LIN {X 74.035,Y -43.514,Z -167.127,A -90.000,B 90.000,C 0.000} C_DIS
LIN {X 73.239,Y -43.520,Z -169.410,A -90.000,B 90.000,C 0.000} C_DIS
LIN {X 72.844,Y -43.519,Z -170.536,A -90.000,B 90.000,C 0.000} C_DIS
LIN {X 72.299,Y -43.524,Z -172.033,A -90.000,B 90.000,C 0.000} C_DIS
LIN {X 72.099,Y -43.529,Z -172.557,A -90.000,B 90.000,C 0.000} C_DIS
LIN {X 71.692,Y -43.549,Z -173.637,A -90.000,B 90.000,C 0.000} C_DIS
LIN {X 71.059,Y -43.555,Z -175.551,A -90.000,B 90.000,C 0.000} C_DIS
LIN {X 70.896,Y -43.570,Z -176.056,A -90.000,B 90.000,C 0.000} C_DIS
LIN {X 70.529,Y -43.551,Z -177.830,A -90.000,B 90.000,C 0.000} C_DIS
LIN {X 70.400,Y -43.548,Z -178.399,A -90.000,B 90.000,C 0.000} C_DIS
LIN {X 70.060,Y -43.525,Z -180.717,A -90.000,B 90.000,C 0.000} C_DIS
LIN {X 70.039,Y -43.519,Z -180.942,A -90.000,B 90.000,C 0.000} C_DIS
LIN {X 69.857,Y -43.488,Z -182.943,A -90.000,B 90.000,C 0.000} C_DIS
LIN {X 69.817,Y -43.471,Z -183.612,A -90.000,B 90.000,C 0.000} C_DIS
LIN {X 69.805,Y -43.466,Z -183.813,A -90.000,B 90.000,C 0.000} C_DIS
LIN {X 69.642,Y -43.421,Z -186.238,A -90.000,B 90.000,C 0.000} C_DIS
LIN {X 69.579,Y -43.400,Z -187.145,A -90.000,B 90.000,C 0.000} C_DIS
LIN {X 69.514,Y -43.379,Z -188.002,A -90.000,B 90.000,C 0.000} C_DIS
LIN {X 69.477,Y -43.368,Z -188.428,A -90.000,B 90.000,C 0.000} C_DIS
LIN {X 69.418,Y -43.357,Z -188.971,A -90.000,B 90.000,C 0.000} C_DIS
LIN {X 69.299,Y -43.324,Z -190.039,A -90.000,B 90.000,C 0.000} C_DIS
LIN {X 69.261,Y -43.308,Z -190.358,A -90.000,B 90.000,C 0.000} C_DIS
LIN {X 69.261,Y -60.000,Z -190.358,A -90.000,B 90.000,C 0.000} C_DIS
LIN {X 59.148,Y -60.000,Z -133.648,A -90.000,B 90.000,C 0.000} C_DIS
LIN {X 59.148,Y -43.308,Z -133.648,A -90.000,B 90.000,C 0.000} C_DIS
LIN {X 59.314,Y -43.330,Z -133.579,A -90.000,B 90.000,C 0.000} C_DIS
LIN {X 59.672,Y -43.381,Z -133.445,A -90.000,B 90.000,C 0.000} C_DIS
LIN {X 60.638,Y -43.533,Z -133.112,A -90.000,B 90.000,C 0.000} C_DIS
LIN {X 61.670,Y -43.677,Z -132.764,A -90.000,B 90.000,C 0.000} C_DIS
LIN {X 61.820,Y -43.698,Z -132.716,A -90.000,B 90.000,C 0.000} C_DIS
LIN {X 61.951,Y -43.718,Z -132.678,A -90.000,B 90.000,C 0.000} C_DIS
LIN {X 62.168,Y -43.758,Z -132.615,A -90.000,B 90.000,C 0.000} C_DIS
LIN {X 62.369,Y -43.796,Z -132.562,A -90.000,B 90.000,C 0.000} C_DIS
LIN {X 62.552,Y -43.831,Z -132.519,A -90.000,B 90.000,C 0.000} C_DIS
LIN {X 62.943,Y -43.909,Z -132.439,A -90.000,B 90.000,C 0.000} C_DIS
LIN {X 63.093,Y -43.940,Z -132.412,A -90.000,B 90.000,C 0.000} C_DIS
LIN {X 63.216,Y -43.967,Z -132.392,A -90.000,B 90.000,C 0.000} C_DIS
LIN {X 63.328,Y -43.991,Z -132.378,A -90.000,B 90.000,C 0.000} C_DIS
LIN {X 63.581,Y -44.028,Z -132.352,A -90.000,B 90.000,C 0.000} C_DIS
LIN {X 63.758,Y -44.054,Z -132.339,A -90.000,B 90.000,C 0.000} C_DIS
LIN {X 64.159,Y -44.115,Z -132.327,A -90.000,B 90.000,C 0.000} C_DIS
LIN {X 64.303,Y -44.138,Z -132.327,A -90.000,B 90.000,C 0.000} C_DIS
LIN {X 65.331,Y -44.306,Z -132.343,A -90.000,B 90.000,C 0.000} C_DIS
LIN {X 65.660,Y -44.358,Z -132.351,A -90.000,B 90.000,C 0.000} C_DIS
LIN {X 65.799,Y -44.369,Z -132.355,A -90.000,B 90.000,C 0.000} C_DIS
LIN {X 65.974,Y -44.379,Z -132.361,A -90.000,B 90.000,C 0.000} C_DIS
LIN {X 66.177,Y -44.391,Z -132.376,A -90.000,B 90.000,C 0.000} C_DIS
LIN {X 66.618,Y -44.418,Z -132.426,A -90.000,B 90.000,C 0.000} C_DIS
LIN {X 66.734,Y -44.426,Z -132.443,A -90.000,B 90.000,C 0.000} C_DIS
LIN {X 67.191,Y -44.459,Z -132.526,A -90.000,B 90.000,C 0.000} C_DIS
LIN {X 67.404,Y -44.474,Z -132.567,A -90.000,B 90.000,C 0.000} C_DIS
LIN {X 67.694,Y -44.496,Z -132.633,A -90.000,B 90.000,C 0.000} C_DIS
LIN {X 67.883,Y -44.509,Z -132.684,A -90.000,B 90.000,C 0.000} C_DIS
LIN {X 68.117,Y -44.524,Z -132.758,A -90.000,B 90.000,C 0.000} C_DIS
LIN {X 68.235,Y -44.524,Z -132.797,A -90.000,B 90.000,C 0.000} C_DIS
LIN {X 69.600,Y -44.469,Z -133.270,A -90.000,B 90.000,C 0.000} C_DIS
LIN {X 69.759,Y -44.463,Z -133.330,A -90.000,B 90.000,C 0.000} C_DIS
LIN {X 70.074,Y -44.451,Z -133.459,A -90.000,B 90.000,C 0.000} C_DIS
LIN {X 70.309,Y -44.443,Z -133.564,A -90.000,B 90.000,C 0.000} C_DIS
LIN {X 70.481,Y -44.437,Z -133.650,A -90.000,B 90.000,C 0.000} C_DIS
LIN {X 70.755,Y -44.429,Z -133.798,A -90.000,B 90.000,C 0.000} C_DIS
LIN {X 70.990,Y -44.420,Z -133.930,A -90.000,B 90.000,C 0.000} C_DIS
LIN {X 71.077,Y -44.411,Z -133.981,A -90.000,B 90.000,C 0.000} C_DIS
LIN {X 71.147,Y -44.402,Z -134.025,A -90.000,B 90.000,C 0.000} C_DIS
LIN {X 71.340,Y -44.376,Z -134.152,A -90.000,B 90.000,C 0.000} C_DIS
LIN {X 71.676,Y -44.334,Z -134.389,A -90.000,B 90.000,C 0.000} C_DIS
LIN {X 71.836,Y -44.314,Z -134.512,A -90.000,B 90.000,C 0.000} C_DIS
LIN {X 72.068,Y -44.286,Z -134.700,A -90.000,B 90.000,C 0.000} C_DIS
LIN {X 72.330,Y -44.255,Z -134.922,A -90.000,B 90.000,C 0.000} C_DIS
LIN {X 72.460,Y -44.240,Z -135.039,A -90.000,B 90.000,C 0.000} C_DIS
LIN {X 72.525,Y -44.233,Z -135.101,A -90.000,B 90.000,C 0.000} C_DIS
LIN {X 72.757,Y -44.206,Z -135.333,A -90.000,B 90.000,C 0.000} C_DIS
LIN {X 73.431,Y -44.132,Z -136.043,A -90.000,B 90.000,C 0.000} C_DIS
LIN {X 73.613,Y -44.113,Z -136.246,A -90.000,B 90.000,C 0.000} C_DIS
LIN {X 73.667,Y -44.107,Z -136.309,A -90.000,B 90.000,C 0.000} C_DIS
LIN {X 73.937,Y -44.080,Z -136.639,A -90.000,B 90.000,C 0.000} C_DIS
LIN {X 74.056,Y -44.065,Z -136.797,A -90.000,B 90.000,C 0.000} C_DIS
LIN {X 74.241,Y -44.043,Z -137.053,A -90.000,B 90.000,C 0.000} C_DIS
LIN {X 74.346,Y -44.031,Z -137.211,A -90.000,B 90.000,C 0.000} C_DIS
LIN {X 74.417,Y -44.017,Z -137.322,A -90.000,B 90.000,C 0.000} C_DIS
LIN {X 74.552,Y -43.991,Z -137.546,A -90.000,B 90.000,C 0.000} C_DIS
LIN {X 74.951,Y -43.916,Z -138.254,A -90.000,B 90.000,C 0.000} C_DIS
LIN {X 75.488,Y -43.810,Z -139.094,A -90.000,B 90.000,C 0.000} C_DIS
LIN {X 75.587,Y -43.791,Z -139.263,A -90.000,B 90.000,C 0.000} C_DIS
LIN {X 75.716,Y -43.767,Z -139.493,A -90.000,B 90.000,C 0.000} C_DIS
LIN {X 75.863,Y -43.740,Z -139.772,A -90.000,B 90.000,C 0.000} C_DIS
LIN {X 76.002,Y -43.711,Z -140.057,A -90.000,B 90.000,C 0.000} C_DIS
LIN {X 76.088,Y -43.694,Z -140.251,A -90.000,B 90.000,C 0.000} C_DIS
LIN {X 76.773,Y -43.558,Z -141.907,A -90.000,B 90.000,C 0.000} C_DIS
LIN {X 76.859,Y -43.541,Z -142.139,A -90.000,B 90.000,C 0.000} C_DIS
LIN {X 77.001,Y -43.514,Z -142.567,A -90.000,B 90.000,C 0.000} C_DIS
LIN {X 77.079,Y -43.501,Z -142.832,A -90.000,B 90.000,C 0.000} C_DIS
LIN {X 77.166,Y -43.485,Z -143.164,A -90.000,B 90.000,C 0.000} C_DIS
LIN {X 77.257,Y -43.465,Z -143.511,A -90.000,B 90.000,C 0.000} C_DIS
LIN {X 77.395,Y -43.429,Z -144.052,A -90.000,B 90.000,C 0.000} C_DIS
LIN {X 77.452,Y -43.415,Z -144.315,A -90.000,B 90.000,C 0.000} C_DIS
LIN {X 77.497,Y -43.400,Z -144.536,A -90.000,B 90.000,C 0.000} C_DIS
LIN {X 77.535,Y -43.387,Z -144.766,A -90.000,B 90.000,C 0.000} C_DIS
LIN {X 77.593,Y -43.367,Z -145.180,A -90.000,B 90.000,C 0.000} C_DIS
LIN {X 77.765,Y -43.308,Z -146.651,A -90.000,B 90.000,C 0.000} C_DIS
LIN {X 77.765,Y -60.000,Z -146.651,A -90.000,B 90.000,C 0.000} C_DIS
LIN {X 61.524,Y -60.000,Z -130.767,A -90.000,B 90.000,C 0.000} C_DIS
LIN {X 61.524,Y -43.308,Z -130.767,A -90.000,B 90.000,C 0.000} C_DIS
LIN {X 61.734,Y -43.351,Z -130.706,A -90.000,B 90.000,C 0.000} C_DIS
LIN {X 61.993,Y -43.405,Z -130.637,A -90.000,B 90.000,C 0.000} C_DIS
LIN {X 62.259,Y -43.462,Z -130.575,A -90.000,B 90.000,C 0.000} C_DIS
LIN {X 62.447,Y -43.502,Z -130.536,A -90.000,B 90.000,C 0.000} C_DIS
LIN {X 62.709,Y -43.555,Z -130.484,A -90.000,B 90.000,C 0.000} C_DIS
LIN {X 62.858,Y -43.586,Z -130.458,A -90.000,B 90.000,C 0.000} C_DIS
LIN {X 63.031,Y -43.623,Z -130.431,A -90.000,B 90.000,C 0.000} C_DIS
LIN {X 63.292,Y -43.680,Z -130.399,A -90.000,B 90.000,C 0.000} C_DIS
LIN {X 63.486,Y -43.722,Z -130.378,A -90.000,B 90.000,C 0.000} C_DIS
LIN {X 63.738,Y -43.779,Z -130.358,A -90.000,B 90.000,C 0.000} C_DIS
LIN {X 64.112,Y -43.865,Z -130.343,A -90.000,B 90.000,C 0.000} C_DIS
LIN {X 64.370,Y -43.920,Z -130.340,A -90.000,B 90.000,C 0.000} C_DIS
LIN {X 64.481,Y -43.944,Z -130.341,A -90.000,B 90.000,C 0.000} C_DIS
LIN {X 65.453,Y -44.105,Z -130.357,A -90.000,B 90.000,C 0.000} C_DIS
LIN {X 65.850,Y -44.167,Z -130.366,A -90.000,B 90.000,C 0.000} C_DIS
LIN {X 66.132,Y -44.203,Z -130.375,A -90.000,B 90.000,C 0.000} C_DIS
LIN {X 66.411,Y -44.240,Z -130.395,A -90.000,B 90.000,C 0.000} C_DIS
LIN {X 66.538,Y -44.257,Z -130.409,A -90.000,B 90.000,C 0.000} C_DIS
LIN {X 66.919,Y -44.283,Z -130.453,A -90.000,B 90.000,C 0.000} C_DIS
LIN {X 67.098,Y -44.297,Z -130.481,A -90.000,B 90.000,C 0.000} C_DIS
LIN {X 67.626,Y -44.341,Z -130.576,A -90.000,B 90.000,C 0.000} C_DIS
LIN {X 67.858,Y -44.361,Z -130.622,A -90.000,B 90.000,C 0.000} C_DIS
LIN {X 68.022,Y -44.375,Z -130.660,A -90.000,B 90.000,C 0.000} C_DIS
LIN {X 68.222,Y -44.388,Z -130.707,A -90.000,B 90.000,C 0.000} C_DIS
LIN {X 68.426,Y -44.400,Z -130.762,A -90.000,B 90.000,C 0.000} C_DIS
LIN {X 68.541,Y -44.400,Z -130.798,A -90.000,B 90.000,C 0.000} C_DIS
LIN {X 68.884,Y -44.388,Z -130.910,A -90.000,B 90.000,C 0.000} C_DIS
LIN {X 70.298,Y -44.340,Z -131.400,A -90.000,B 90.000,C 0.000} C_DIS
LIN {X 70.457,Y -44.335,Z -131.460,A -90.000,B 90.000,C 0.000} C_DIS
LIN {X 70.885,Y -44.322,Z -131.635,A -90.000,B 90.000,C 0.000} C_DIS
LIN {X 71.191,Y -44.306,Z -131.775,A -90.000,B 90.000,C 0.000} C_DIS
LIN {X 71.340,Y -44.296,Z -131.849,A -90.000,B 90.000,C 0.000} C_DIS
LIN {X 71.465,Y -44.279,Z -131.915,A -90.000,B 90.000,C 0.000} C_DIS
LIN {X 71.831,Y -44.230,Z -132.119,A -90.000,B 90.000,C 0.000} C_DIS
LIN {X 72.000,Y -44.207,Z -132.216,A -90.000,B 90.000,C 0.000} C_DIS
LIN {X 72.222,Y -44.177,Z -132.353,A -90.000,B 90.000,C 0.000} C_DIS
LIN {X 72.464,Y -44.146,Z -132.514,A -90.000,B 90.000,C 0.000} C_DIS
LIN {X 72.800,Y -44.101,Z -132.751,A -90.000,B 90.000,C 0.000} C_DIS
LIN {X 73.023,Y -44.072,Z -132.920,A -90.000,B 90.000,C 0.000} C_DIS
LIN {X 73.302,Y -44.035,Z -133.146,A -90.000,B 90.000,C 0.000} C_DIS
LIN {X 73.592,Y -43.997,Z -133.391,A -90.000,B 90.000,C 0.000} C_DIS
LIN {X 73.806,Y -43.969,Z -133.585,A -90.000,B 90.000,C 0.000} C_DIS
LIN {X 73.910,Y -43.956,Z -133.685,A -90.000,B 90.000,C 0.000} C_DIS
LIN {X 74.184,Y -43.923,Z -133.960,A -90.000,B 90.000,C 0.000} C_DIS
LIN {X 74.595,Y -43.865,Z -134.396,A -90.000,B 90.000,C 0.000} C_DIS
LIN {X 74.888,Y -43.805,Z -134.712,A -90.000,B 90.000,C 0.000} C_DIS
LIN {X 75.121,Y -43.758,Z -134.980,A -90.000,B 90.000,C 0.000} C_DIS
LIN {X 75.440,Y -43.694,Z -135.378,A -90.000,B 90.000,C 0.000} C_DIS
LIN {X 75.625,Y -43.658,Z -135.626,A -90.000,B 90.000,C 0.000} C_DIS
LIN {X 75.852,Y -43.614,Z -135.949,A -90.000,B 90.000,C 0.000} C_DIS
LIN {X 76.064,Y -43.574,Z -136.278,A -90.000,B 90.000,C 0.000} C_DIS
LIN {X 76.230,Y -43.543,Z -136.553,A -90.000,B 90.000,C 0.000} C_DIS
LIN {X 76.600,Y -43.471,Z -137.212,A -90.000,B 90.000,C 0.000} C_DIS
LIN {X 77.143,Y -43.361,Z -138.065,A -90.000,B 90.000,C 0.000} C_DIS
LIN {X 77.193,Y -43.351,Z -138.149,A -90.000,B 90.000,C 0.000} C_DIS
LIN {X 77.269,Y -43.336,Z -138.281,A -90.000,B 90.000,C 0.000} C_DIS
LIN {X 77.411,Y -43.308,Z -138.537,A -90.000,B 90.000,C 0.000} C_DIS
LIN {X 77.411,Y -60.000,Z -138.537,A -90.000,B 90.000,C 0.000} C_DIS
LIN {X 63.075,Y -60.000,Z -128.445,A -90.000,B 90.000,C 0.000} C_DIS
LIN {X 63.075,Y -43.308,Z -128.445,A -90.000,B 90.000,C 0.000} C_DIS
LIN {X 63.336,Y -43.368,Z -128.415,A -90.000,B 90.000,C 0.000} C_DIS
LIN {X 63.636,Y -43.439,Z -128.390,A -90.000,B 90.000,C 0.000} C_DIS
LIN {X 63.851,Y -43.491,Z -128.378,A -90.000,B 90.000,C 0.000} C_DIS
LIN {X 64.153,Y -43.564,Z -128.366,A -90.000,B 90.000,C 0.000} C_DIS
LIN {X 64.400,Y -43.623,Z -128.362,A -90.000,B 90.000,C 0.000} C_DIS
LIN {X 64.687,Y -43.684,Z -128.365,A -90.000,B 90.000,C 0.000} C_DIS
LIN {X 65.007,Y -43.746,Z -128.368,A -90.000,B 90.000,C 0.000} C_DIS
LIN {X 65.868,Y -43.902,Z -128.382,A -90.000,B 90.000,C 0.000} C_DIS
LIN {X 66.228,Y -43.947,Z -128.394,A -90.000,B 90.000,C 0.000} C_DIS
LIN {X 66.527,Y -43.986,Z -128.414,A -90.000,B 90.000,C 0.000} C_DIS
LIN {X 66.866,Y -44.031,Z -128.447,A -90.000,B 90.000,C 0.000} C_DIS
LIN {X 67.235,Y -44.081,Z -128.489,A -90.000,B 90.000,C 0.000} C_DIS
LIN {X 67.485,Y -44.113,Z -128.527,A -90.000,B 90.000,C 0.000} C_DIS
LIN {X 67.620,Y -44.131,Z -128.551,A -90.000,B 90.000,C 0.000} C_DIS
LIN {X 67.973,Y -44.168,Z -128.614,A -90.000,B 90.000,C 0.000} C_DIS
LIN {X 68.094,Y -44.180,Z -128.637,A -90.000,B 90.000,C 0.000} C_DIS
LIN {X 68.316,Y -44.192,Z -128.683,A -90.000,B 90.000,C 0.000} C_DIS
LIN {X 68.672,Y -44.204,Z -128.767,A -90.000,B 90.000,C 0.000} C_DIS
LIN {X 69.013,Y -44.216,Z -128.859,A -90.000,B 90.000,C 0.000} C_DIS
LIN {X 69.252,Y -44.226,Z -128.934,A -90.000,B 90.000,C 0.000} C_DIS
LIN {X 69.461,Y -44.225,Z -129.002,A -90.000,B 90.000,C 0.000} C_DIS
LIN {X 70.377,Y -44.218,Z -129.316,A -90.000,B 90.000,C 0.000} C_DIS
LIN {X 71.025,Y -44.204,Z -129.542,A -90.000,B 90.000,C 0.000} C_DIS
LIN {X 71.208,Y -44.197,Z -129.612,A -90.000,B 90.000,C 0.000} C_DIS
LIN {X 71.422,Y -44.186,Z -129.700,A -90.000,B 90.000,C 0.000} C_DIS
LIN {X 71.539,Y -44.174,Z -129.748,A -90.000,B 90.000,C 0.000} C_DIS
LIN {X 71.705,Y -44.153,Z -129.819,A -90.000,B 90.000,C 0.000} C_DIS
LIN {X 72.069,Y -44.107,Z -129.989,A -90.000,B 90.000,C 0.000} C_DIS
LIN {X 72.247,Y -44.085,Z -130.079,A -90.000,B 90.000,C 0.000} C_DIS
LIN {X 72.410,Y -44.065,Z -130.166,A -90.000,B 90.000,C 0.000} C_DIS
LIN {X 72.798,Y -44.018,Z -130.382,A -90.000,B 90.000,C 0.000} C_DIS
LIN {X 73.025,Y -43.989,Z -130.513,A -90.000,B 90.000,C 0.000} C_DIS
LIN {X 73.302,Y -43.953,Z -130.685,A -90.000,B 90.000,C 0.000} C_DIS
LIN {X 73.587,Y -43.916,Z -130.876,A -90.000,B 90.000,C 0.000} C_DIS
LIN {X 73.924,Y -43.873,Z -131.113,A -90.000,B 90.000,C 0.000} C_DIS
LIN {X 74.260,Y -43.831,Z -131.367,A -90.000,B 90.000,C 0.000} C_DIS
LIN {X 74.393,Y -43.814,Z -131.474,A -90.000,B 90.000,C 0.000} C_DIS
LIN {X 74.563,Y -43.786,Z -131.614,A -90.000,B 90.000,C 0.000} C_DIS
LIN {X 74.845,Y -43.739,Z -131.854,A -90.000,B 90.000,C 0.000} C_DIS
LIN {X 75.092,Y -43.688,Z -132.079,A -90.000,B 90.000,C 0.000} C_DIS
LIN {X 75.217,Y -43.662,Z -132.198,A -90.000,B 90.000,C 0.000} C_DIS
LIN {X 75.318,Y -43.641,Z -132.299,A -90.000,B 90.000,C 0.000} C_DIS
LIN {X 75.594,Y -43.585,Z -132.583,A -90.000,B 90.000,C 0.000} C_DIS
LIN {X 76.088,Y -43.484,Z -133.115,A -90.000,B 90.000,C 0.000} C_DIS
LIN {X 76.297,Y -43.439,Z -133.341,A -90.000,B 90.000,C 0.000} C_DIS
LIN {X 76.572,Y -43.379,Z -133.657,A -90.000,B 90.000,C 0.000} C_DIS
LIN {X 76.904,Y -43.308,Z -134.070,A -90.000,B 90.000,C 0.000} C_DIS
LIN {X 76.904,Y -60.000,Z -134.070,A -90.000,B 90.000,C 0.000} C_DIS
LIN {X 64.689,Y -60.000,Z -126.398,A -90.000,B 90.000,C 0.000} C_DIS
LIN {X 64.689,Y -43.308,Z -126.398,A -90.000,B 90.000,C 0.000} C_DIS
LIN {X 66.152,Y -43.583,Z -126.420,A -90.000,B 90.000,C 0.000} C_DIS
LIN {X 66.403,Y -43.631,Z -126.426,A -90.000,B 90.000,C 0.000} C_DIS
LIN {X 66.782,Y -43.704,Z -126.450,A -90.000,B 90.000,C 0.000} C_DIS
LIN {X 67.055,Y -43.742,Z -126.477,A -90.000,B 90.000,C 0.000} C_DIS
LIN {X 67.331,Y -43.770,Z -126.508,A -90.000,B 90.000,C 0.000} C_DIS
LIN {X 67.571,Y -43.789,Z -126.539,A -90.000,B 90.000,C 0.000} C_DIS
LIN {X 68.003,Y -43.828,Z -126.611,A -90.000,B 90.000,C 0.000} C_DIS
LIN {X 68.496,Y -43.873,Z -126.702,A -90.000,B 90.000,C 0.000} C_DIS
LIN {X 68.692,Y -43.891,Z -126.741,A -90.000,B 90.000,C 0.000} C_DIS
LIN {X 69.128,Y -43.930,Z -126.839,A -90.000,B 90.000,C 0.000} C_DIS
LIN {X 69.209,Y -43.937,Z -126.859,A -90.000,B 90.000,C 0.000} C_DIS
LIN {X 69.614,Y -43.953,Z -126.970,A -90.000,B 90.000,C 0.000} C_DIS
LIN {X 70.103,Y -43.974,Z -127.125,A -90.000,B 90.000,C 0.000} C_DIS
LIN {X 70.834,Y -44.007,Z -127.371,A -90.000,B 90.000,C 0.000} C_DIS
LIN {X 71.029,Y -44.007,Z -127.438,A -90.000,B 90.000,C 0.000} C_DIS
LIN {X 71.236,Y -43.996,Z -127.510,A -90.000,B 90.000,C 0.000} C_DIS
LIN {X 71.741,Y -43.954,Z -127.691,A -90.000,B 90.000,C 0.000} C_DIS
LIN {X 71.993,Y -43.935,Z -127.791,A -90.000,B 90.000,C 0.000} C_DIS
LIN {X 72.442,Y -43.901,Z -127.977,A -90.000,B 90.000,C 0.000} C_DIS
LIN {X 72.538,Y -43.894,Z -128.019,A -90.000,B 90.000,C 0.000} C_DIS
LIN {X 72.944,Y -43.865,Z -128.207,A -90.000,B 90.000,C 0.000} C_DIS
LIN {X 73.019,Y -43.859,Z -128.244,A -90.000,B 90.000,C 0.000} C_DIS
LIN {X 73.154,Y -43.845,Z -128.313,A -90.000,B 90.000,C 0.000} C_DIS
LIN {X 73.353,Y -43.823,Z -128.419,A -90.000,B 90.000,C 0.000} C_DIS
LIN {X 73.769,Y -43.779,Z -128.650,A -90.000,B 90.000,C 0.000} C_DIS
LIN {X 73.996,Y -43.755,Z -128.780,A -90.000,B 90.000,C 0.000} C_DIS
LIN {X 74.383,Y -43.716,Z -129.019,A -90.000,B 90.000,C 0.000} C_DIS
LIN {X 74.578,Y -43.693,Z -129.149,A -90.000,B 90.000,C 0.000} C_DIS
LIN {X 74.667,Y -43.682,Z -129.209,A -90.000,B 90.000,C 0.000} C_DIS
LIN {X 74.781,Y -43.666,Z -129.288,A -90.000,B 90.000,C 0.000} C_DIS
LIN {X 75.006,Y -43.629,Z -129.449,A -90.000,B 90.000,C 0.000} C_DIS
LIN {X 75.127,Y -43.605,Z -129.537,A -90.000,B 90.000,C 0.000} C_DIS
LIN {X 75.483,Y -43.536,Z -129.812,A -90.000,B 90.000,C 0.000} C_DIS
LIN {X 75.812,Y -43.473,Z -130.084,A -90.000,B 90.000,C 0.000} C_DIS
LIN {X 76.128,Y -43.412,Z -130.355,A -90.000,B 90.000,C 0.000} C_DIS
LIN {X 76.418,Y -43.355,Z -130.619,A -90.000,B 90.000,C 0.000} C_DIS
LIN {X 76.624,Y -43.312,Z -130.819,A -90.000,B 90.000,C 0.000} C_DIS
LIN {X 76.640,Y -43.308,Z -130.834,A -90.000,B 90.000,C 0.000} C_DIS
LIN {X 76.640,Y -60.000,Z -130.834,A -90.000,B 90.000,C 0.000} C_DIS
LIN {X 66.732,Y -60.000,Z -124.475,A -90.000,B 90.000,C 0.000} C_DIS
LIN {X 66.732,Y -43.308,Z -124.475,A -90.000,B 90.000,C 0.000} C_DIS
LIN {X 66.961,Y -43.334,Z -124.493,A -90.000,B 90.000,C 0.000} C_DIS
LIN {X 67.315,Y -43.370,Z -124.529,A -90.000,B 90.000,C 0.000} C_DIS
LIN {X 67.834,Y -43.425,Z -124.590,A -90.000,B 90.000,C 0.000} C_DIS
LIN {X 68.028,Y -43.444,Z -124.620,A -90.000,B 90.000,C 0.000} C_DIS
LIN {X 68.449,Y -43.488,Z -124.691,A -90.000,B 90.000,C 0.000} C_DIS
LIN {X 68.912,Y -43.538,Z -124.775,A -90.000,B 90.000,C 0.000} C_DIS
LIN {X 69.151,Y -43.564,Z -124.823,A -90.000,B 90.000,C 0.000} C_DIS
LIN {X 69.626,Y -43.617,Z -124.928,A -90.000,B 90.000,C 0.000} C_DIS
LIN {X 69.825,Y -43.640,Z -124.978,A -90.000,B 90.000,C 0.000} C_DIS
LIN {X 70.032,Y -43.658,Z -125.033,A -90.000,B 90.000,C 0.000} C_DIS
LIN {X 70.227,Y -43.666,Z -125.088,A -90.000,B 90.000,C 0.000} C_DIS
LIN {X 70.645,Y -43.678,Z -125.221,A -90.000,B 90.000,C 0.000} C_DIS
LIN {X 70.927,Y -43.673,Z -125.317,A -90.000,B 90.000,C 0.000} C_DIS
LIN {X 71.626,Y -43.661,Z -125.560,A -90.000,B 90.000,C 0.000} C_DIS
LIN {X 72.431,Y -43.641,Z -125.840,A -90.000,B 90.000,C 0.000} C_DIS
LIN {X 72.761,Y -43.635,Z -125.968,A -90.000,B 90.000,C 0.000} C_DIS
LIN {X 73.001,Y -43.627,Z -126.066,A -90.000,B 90.000,C 0.000} C_DIS
LIN {X 73.292,Y -43.606,Z -126.189,A -90.000,B 90.000,C 0.000} C_DIS
LIN {X 73.813,Y -43.571,Z -126.430,A -90.000,B 90.000,C 0.000} C_DIS
LIN {X 74.103,Y -43.553,Z -126.576,A -90.000,B 90.000,C 0.000} C_DIS
LIN {X 74.303,Y -43.539,Z -126.682,A -90.000,B 90.000,C 0.000} C_DIS
LIN {X 74.684,Y -43.506,Z -126.892,A -90.000,B 90.000,C 0.000} C_DIS
LIN {X 74.738,Y -43.501,Z -126.922,A -90.000,B 90.000,C 0.000} C_DIS
LIN {X 74.968,Y -43.474,Z -127.055,A -90.000,B 90.000,C 0.000} C_DIS
LIN {X 75.440,Y -43.401,Z -127.351,A -90.000,B 90.000,C 0.000} C_DIS
LIN {X 75.757,Y -43.353,Z -127.564,A -90.000,B 90.000,C 0.000} C_DIS
LIN {X 76.052,Y -43.308,Z -127.773,A -90.000,B 90.000,C 0.000} C_DIS
LIN {X 76.052,Y -60.000,Z -127.773,A -90.000,B 90.000,C 0.000} C_DIS
LIN {X -72.201,Y -60.000,Z -243.561,A -90.000,B 90.000,C 0.000} C_DIS
LIN {X -72.201,Y -43.308,Z -243.561,A -90.000,B 90.000,C 0.000} C_DIS
LIN {X -70.197,Y -43.308,Z -242.446,A -90.000,B 90.000,C 0.000} C_DIS
LIN {X -67.566,Y -43.308,Z -241.012,A -90.000,B 90.000,C 0.000} C_DIS
LIN {X -67.295,Y -43.308,Z -240.867,A -90.000,B 90.000,C 0.000} C_DIS
LIN {X -65.307,Y -43.308,Z -239.852,A -90.000,B 90.000,C 0.000} C_DIS
LIN {X -58.869,Y -43.308,Z -236.542,A -90.000,B 90.000,C 0.000} C_DIS
LIN {X -56.444,Y -43.308,Z -235.343,A -90.000,B 90.000,C 0.000} C_DIS
LIN {X -51.943,Y -43.308,Z -233.181,A -90.000,B 90.000,C 0.000} C_DIS
LIN {X -50.867,Y -43.308,Z -232.682,A -90.000,B 90.000,C 0.000} C_DIS
LIN {X -45.478,Y -43.308,Z -230.277,A -90.000,B 90.000,C 0.000} C_DIS
LIN {X -41.771,Y -43.308,Z -228.705,A -90.000,B 90.000,C 0.000} C_DIS
LIN {X -39.806,Y -43.308,Z -227.846,A -90.000,B 90.000,C 0.000} C_DIS
LIN {X -36.653,Y -43.308,Z -226.535,A -90.000,B 90.000,C 0.000} C_DIS
LIN {X -36.468,Y -43.308,Z -226.460,A -90.000,B 90.000,C 0.000} C_DIS
LIN {X -34.673,Y -43.308,Z -225.787,A -90.000,B 90.000,C 0.000} C_DIS
LIN {X -33.189,Y -43.308,Z -225.268,A -90.000,B 90.000,C 0.000} C_DIS
LIN {X -30.217,Y -43.308,Z -224.139,A -90.000,B 90.000,C 0.000} C_DIS
LIN {X -25.730,Y -43.308,Z -222.512,A -90.000,B 90.000,C 0.000} C_DIS
LIN {X -25.382,Y -43.308,Z -222.367,A -90.000,B 90.000,C 0.000} C_DIS
LIN {X -24.084,Y -43.308,Z -221.960,A -90.000,B 90.000,C 0.000} C_DIS
LIN {X -18.835,Y -43.308,Z -220.340,A -90.000,B 90.000,C 0.000} C_DIS
LIN {X -17.915,Y -43.308,Z -219.996,A -90.000,B 90.000,C 0.000} C_DIS
LIN {X -16.736,Y -43.308,Z -219.532,A -90.000,B 90.000,C 0.000} C_DIS
LIN {X -16.505,Y -43.308,Z -219.480,A -90.000,B 90.000,C 0.000} C_DIS
LIN {X -14.654,Y -43.308,Z -219.084,A -90.000,B 90.000,C 0.000} C_DIS
LIN {X -12.352,Y -43.308,Z -218.525,A -90.000,B 90.000,C 0.000} C_DIS
LIN {X -11.727,Y -43.308,Z -218.326,A -90.000,B 90.000,C 0.000} C_DIS
LIN {X -11.012,Y -43.308,Z -218.058,A -90.000,B 90.000,C 0.000} C_DIS
LIN {X -9.958,Y -43.308,Z -217.682,A -90.000,B 90.000,C 0.000} C_DIS
LIN {X -9.784,Y -43.308,Z -217.639,A -90.000,B 90.000,C 0.000} C_DIS
LIN {X -8.428,Y -43.308,Z -217.535,A -90.000,B 90.000,C 0.000} C_DIS
LIN {X -6.386,Y -43.308,Z -217.134,A -90.000,B 90.000,C 0.000} C_DIS
LIN {X -5.896,Y -43.308,Z -217.008,A -90.000,B 90.000,C 0.000} C_DIS
LIN {X -5.217,Y -43.308,Z -216.719,A -90.000,B 90.000,C 0.000} C_DIS
LIN {X -5.043,Y -43.308,Z -216.676,A -90.000,B 90.000,C 0.000} C_DIS
LIN {X -4.392,Y -43.308,Z -216.567,A -90.000,B 90.000,C 0.000} C_DIS
LIN {X -3.000,Y -43.308,Z -216.642,A -90.000,B 90.000,C 0.000} C_DIS
LIN {X -0.702,Y -43.308,Z -215.900,A -90.000,B 90.000,C 0.000} C_DIS
LIN {X 0.084,Y -43.308,Z -215.465,A -90.000,B 90.000,C 0.000} C_DIS
LIN {X 0.166,Y -43.308,Z -215.431,A -90.000,B 90.000,C 0.000} C_DIS
LIN {X 2.161,Y -43.308,Z -215.036,A -90.000,B 90.000,C 0.000} C_DIS
LIN {X 3.987,Y -43.308,Z -213.191,A -90.000,B 90.000,C 0.000} C_DIS
LIN {X 4.915,Y -43.308,Z -212.335,A -90.000,B 90.000,C 0.000} C_DIS
LIN {X 7.001,Y -43.308,Z -209.239,A -90.000,B 90.000,C 0.000} C_DIS
LIN {X 8.267,Y -43.308,Z -207.502,A -90.000,B 90.000,C 0.000} C_DIS
LIN {X 9.588,Y -43.308,Z -205.135,A -90.000,B 90.000,C 0.000} C_DIS
LIN {X 11.591,Y -43.308,Z -201.754,A -90.000,B 90.000,C 0.000} C_DIS
LIN {X 11.879,Y -43.308,Z -201.170,A -90.000,B 90.000,C 0.000} C_DIS
LIN {X 12.860,Y -43.308,Z -199.267,A -90.000,B 90.000,C 0.000} C_DIS
LIN {X 12.973,Y -43.308,Z -199.063,A -90.000,B 90.000,C 0.000} C_DIS
LIN {X 14.251,Y -43.308,Z -196.849,A -90.000,B 90.000,C 0.000} C_DIS
LIN {X 14.395,Y -43.308,Z -196.621,A -90.000,B 90.000,C 0.000} C_DIS
LIN {X 14.494,Y -43.308,Z -196.440,A -90.000,B 90.000,C 0.000} C_DIS
LIN {X 16.439,Y -43.308,Z -193.001,A -90.000,B 90.000,C 0.000} C_DIS
LIN {X 16.591,Y -43.308,Z -192.764,A -90.000,B 90.000,C 0.000} C_DIS
LIN {X 17.389,Y -43.308,Z -191.553,A -90.000,B 90.000,C 0.000} C_DIS
LIN {X 18.724,Y -43.308,Z -189.307,A -90.000,B 90.000,C 0.000} C_DIS
LIN {X 18.877,Y -43.308,Z -189.070,A -90.000,B 90.000,C 0.000} C_DIS
LIN {X 20.089,Y -43.308,Z -187.402,A -90.000,B 90.000,C 0.000} C_DIS
LIN {X 21.154,Y -43.308,Z -185.789,A -90.000,B 90.000,C 0.000} C_DIS
LIN {X 22.609,Y -43.308,Z -183.933,A -90.000,B 90.000,C 0.000} C_DIS
LIN {X 23.352,Y -43.308,Z -183.055,A -90.000,B 90.000,C 0.000} C_DIS
LIN {X 25.478,Y -43.308,Z -180.625,A -90.000,B 90.000,C 0.000} C_DIS
LIN {X 25.659,Y -43.308,Z -180.429,A -90.000,B 90.000,C 0.000} C_DIS
LIN {X 26.382,Y -43.308,Z -179.590,A -90.000,B 90.000,C 0.000} C_DIS
LIN {X 27.500,Y -43.308,Z -178.328,A -90.000,B 90.000,C 0.000} C_DIS
LIN {X 29.081,Y -43.308,Z -176.415,A -90.000,B 90.000,C 0.000} C_DIS
LIN {X 29.170,Y -43.308,Z -176.311,A -90.000,B 90.000,C 0.000} C_DIS
LIN {X 30.538,Y -43.308,Z -174.479,A -90.000,B 90.000,C 0.000} C_DIS
LIN {X 30.846,Y -43.308,Z -174.006,A -90.000,B 90.000,C 0.000} C_DIS
LIN {X 31.945,Y -43.308,Z -172.389,A -90.000,B 90.000,C 0.000} C_DIS
LIN {X 32.512,Y -43.308,Z -171.446,A -90.000,B 90.000,C 0.000} C_DIS
LIN {X 33.294,Y -43.308,Z -170.201,A -90.000,B 90.000,C 0.000} C_DIS
LIN {X 34.127,Y -43.308,Z -168.743,A -90.000,B 90.000,C 0.000} C_DIS
LIN {X 34.629,Y -43.308,Z -167.893,A -90.000,B 90.000,C 0.000} C_DIS
LIN {X 35.746,Y -43.308,Z -165.874,A -90.000,B 90.000,C 0.000} C_DIS
LIN {X 36.002,Y -43.308,Z -165.419,A -90.000,B 90.000,C 0.000} C_DIS
LIN {X 36.626,Y -43.308,Z -164.255,A -90.000,B 90.000,C 0.000} C_DIS
LIN {X 37.502,Y -43.308,Z -162.660,A -90.000,B 90.000,C 0.000} C_DIS
LIN {X 37.851,Y -43.308,Z -161.997,A -90.000,B 90.000,C 0.000} C_DIS
LIN {X 39.094,Y -43.308,Z -159.676,A -90.000,B 90.000,C 0.000} C_DIS
LIN {X 40.684,Y -43.308,Z -156.625,A -90.000,B 90.000,C 0.000} C_DIS
LIN {X 40.894,Y -43.308,Z -156.211,A -90.000,B 90.000,C 0.000} C_DIS
LIN {X 41.543,Y -43.308,Z -154.967,A -90.000,B 90.000,C 0.000} C_DIS
LIN {X 42.234,Y -43.308,Z -153.680,A -90.000,B 90.000,C 0.000} C_DIS
LIN {X 42.920,Y -43.308,Z -152.432,A -90.000,B 90.000,C 0.000} C_DIS
LIN {X 43.573,Y -43.308,Z -151.270,A -90.000,B 90.000,C 0.000} C_DIS
LIN {X 43.867,Y -43.308,Z -150.764,A -90.000,B 90.000,C 0.000} C_DIS
LIN {X 44.789,Y -43.308,Z -149.213,A -90.000,B 90.000,C 0.000} C_DIS
LIN {X 44.959,Y -43.308,Z -148.942,A -90.000,B 90.000,C 0.000} C_DIS
LIN {X 45.969,Y -43.308,Z -147.351,A -90.000,B 90.000,C 0.000} C_DIS
LIN {X 46.279,Y -43.308,Z -146.873,A -90.000,B 90.000,C 0.000} C_DIS
LIN {X 46.774,Y -43.308,Z -146.176,A -90.000,B 90.000,C 0.000} C_DIS
LIN {X 48.432,Y -43.308,Z -144.008,A -90.000,B 90.000,C 0.000} C_DIS
LIN {X 49.205,Y -43.308,Z -143.087,A -90.000,B 90.000,C 0.000} C_DIS
LIN {X 49.415,Y -43.308,Z -142.846,A -90.000,B 90.000,C 0.000} C_DIS
LIN {X 50.239,Y -43.308,Z -141.934,A -90.000,B 90.000,C 0.000} C_DIS
LIN {X 51.239,Y -43.308,Z -140.916,A -90.000,B 90.000,C 0.000} C_DIS
LIN {X 51.610,Y -43.308,Z -140.548,A -90.000,B 90.000,C 0.000} C_DIS
LIN {X 52.912,Y -43.308,Z -139.287,A -90.000,B 90.000,C 0.000} C_DIS
LIN {X 54.102,Y -43.308,Z -138.165,A -90.000,B 90.000,C 0.000} C_DIS
LIN {X 54.622,Y -43.308,Z -137.732,A -90.000,B 90.000,C 0.000} C_DIS
LIN {X 55.187,Y -43.308,Z -137.243,A -90.000,B 90.000,C 0.000} C_DIS
LIN {X 56.337,Y -43.308,Z -136.216,A -90.000,B 90.000,C 0.000} C_DIS
LIN {X 57.534,Y -43.308,Z -135.123,A -90.000,B 90.000,C 0.000} C_DIS
LIN {X 57.997,Y -43.308,Z -134.755,A -90.000,B 90.000,C 0.000} C_DIS
LIN {X 58.398,Y -43.308,Z -134.402,A -90.000,B 90.000,C 0.000} C_DIS
LIN {X 59.623,Y -43.308,Z -133.171,A -90.000,B 90.000,C 0.000} C_DIS
LIN {X 60.644,Y -43.308,Z -132.097,A -90.000,B 90.000,C 0.000} C_DIS
LIN {X 62.211,Y -43.308,Z -129.729,A -90.000,B 90.000,C 0.000} C_DIS
LIN {X 63.036,Y -43.308,Z -128.509,A -90.000,B 90.000,C 0.000} C_DIS
LIN {X 63.714,Y -43.308,Z -127.403,A -90.000,B 90.000,C 0.000} C_DIS
LIN {X 63.869,Y -43.308,Z -127.225,A -90.000,B 90.000,C 0.000} C_DIS
LIN {X 64.446,Y -43.308,Z -126.690,A -90.000,B 90.000,C 0.000} C_DIS
LIN {X 65.704,Y -43.308,Z -125.179,A -90.000,B 90.000,C 0.000} C_DIS
LIN {X 65.763,Y -43.308,Z -125.111,A -90.000,B 90.000,C 0.000} C_DIS
LIN {X 65.773,Y -43.308,Z -125.096,A -90.000,B 90.000,C 0.000} C_DIS
LIN {X 65.929,Y -43.308,Z -124.918,A -90.000,B 90.000,C 0.000} C_DIS
LIN {X 66.118,Y -43.308,Z -124.776,A -90.000,B 90.000,C 0.000} C_DIS
LIN {X 68.592,Y -43.308,Z -123.565,A -90.000,B 90.000,C 0.000} C_DIS
LIN {X 69.037,Y -43.308,Z -123.227,A -90.000,B 90.000,C 0.000} C_DIS
LIN {X 69.193,Y -43.308,Z -123.139,A -90.000,B 90.000,C 0.000} C_DIS
LIN {X 69.367,Y -43.308,Z -123.096,A -90.000,B 90.000,C 0.000} C_DIS
LIN {X 69.546,Y -43.308,Z -123.103,A -90.000,B 90.000,C 0.000} C_DIS
LIN {X 69.724,Y -43.308,Z -123.121,A -90.000,B 90.000,C 0.000} C_DIS
LIN {X 69.947,Y -43.308,Z -123.166,A -90.000,B 90.000,C 0.000} C_DIS
LIN {X 70.670,Y -43.308,Z -123.321,A -90.000,B 90.000,C 0.000} C_DIS
LIN {X 71.533,Y -43.308,Z -123.528,A -90.000,B 90.000,C 0.000} C_DIS
LIN {X 71.704,Y -43.308,Z -123.584,A -90.000,B 90.000,C 0.000} C_DIS
LIN {X 73.700,Y -43.308,Z -124.329,A -90.000,B 90.000,C 0.000} C_DIS
LIN {X 73.848,Y -43.308,Z -124.430,A -90.000,B 90.000,C 0.000} C_DIS
LIN {X 74.312,Y -43.308,Z -124.766,A -90.000,B 90.000,C 0.000} C_DIS
LIN {X 74.435,Y -43.308,Z -124.892,A -90.000,B 90.000,C 0.000} C_DIS
LIN {X 74.594,Y -43.308,Z -125.067,A -90.000,B 90.000,C 0.000} C_DIS
LIN {X 75.516,Y -43.308,Z -126.428,A -90.000,B 90.000,C 0.000} C_DIS
LIN {X 75.636,Y -43.308,Z -126.633,A -90.000,B 90.000,C 0.000} C_DIS
LIN {X 75.802,Y -43.308,Z -127.073,A -90.000,B 90.000,C 0.000} C_DIS
LIN {X 76.214,Y -43.308,Z -128.224,A -90.000,B 90.000,C 0.000} C_DIS
LIN {X 76.287,Y -43.308,Z -128.449,A -90.000,B 90.000,C 0.000} C_DIS
LIN {X 76.428,Y -43.308,Z -129.206,A -90.000,B 90.000,C 0.000} C_DIS
LIN {X 76.586,Y -43.308,Z -130.259,A -90.000,B 90.000,C 0.000} C_DIS
LIN {X 76.611,Y -43.308,Z -130.494,A -90.000,B 90.000,C 0.000} C_DIS
LIN {X 76.700,Y -43.308,Z -131.563,A -90.000,B 90.000,C 0.000} C_DIS
LIN {X 76.800,Y -43.308,Z -132.522,A -90.000,B 90.000,C 0.000} C_DIS
LIN {X 76.896,Y -43.308,Z -133.990,A -90.000,B 90.000,C 0.000} C_DIS
LIN {X 77.113,Y -43.308,Z -136.028,A -90.000,B 90.000,C 0.000} C_DIS
LIN {X 77.199,Y -43.308,Z -136.610,A -90.000,B 90.000,C 0.000} C_DIS
LIN {X 77.540,Y -43.308,Z -139.710,A -90.000,B 90.000,C 0.000} C_DIS
LIN {X 77.565,Y -43.308,Z -140.062,A -90.000,B 90.000,C 0.000} C_DIS
LIN {X 77.708,Y -43.308,Z -142.338,A -90.000,B 90.000,C 0.000} C_DIS
LIN {X 77.751,Y -43.308,Z -143.528,A -90.000,B 90.000,C 0.000} C_DIS
LIN {X 77.748,Y -43.308,Z -143.767,A -90.000,B 90.000,C 0.000} C_DIS
LIN {X 77.769,Y -43.308,Z -147.220,A -90.000,B 90.000,C 0.000} C_DIS
LIN {X 77.719,Y -43.308,Z -148.311,A -90.000,B 90.000,C 0.000} C_DIS
LIN {X 77.615,Y -43.308,Z -151.150,A -90.000,B 90.000,C 0.000} C_DIS
LIN {X 77.459,Y -43.308,Z -152.911,A -90.000,B 90.000,C 0.000} C_DIS
LIN {X 77.287,Y -43.308,Z -154.979,A -90.000,B 90.000,C 0.000} C_DIS
LIN {X 76.963,Y -43.308,Z -157.286,A -90.000,B 90.000,C 0.000} C_DIS
LIN {X 76.759,Y -43.308,Z -158.759,A -90.000,B 90.000,C 0.000} C_DIS
LIN {X 76.712,Y -43.308,Z -159.037,A -90.000,B 90.000,C 0.000} C_DIS
LIN {X 75.958,Y -43.308,Z -162.700,A -90.000,B 90.000,C 0.000} C_DIS
LIN {X 74.948,Y -43.308,Z -166.181,A -90.000,B 90.000,C 0.000} C_DIS
LIN {X 73.817,Y -43.308,Z -169.493,A -90.000,B 90.000,C 0.000} C_DIS
LIN {X 72.699,Y -43.308,Z -172.646,A -90.000,B 90.000,C 0.000} C_DIS
LIN {X 71.731,Y -43.308,Z -175.652,A -90.000,B 90.000,C 0.000} C_DIS
LIN {X 71.045,Y -43.308,Z -178.529,A -90.000,B 90.000,C 0.000} C_DIS
LIN {X 70.609,Y -43.308,Z -181.028,A -90.000,B 90.000,C 0.000} C_DIS
LIN {X 70.320,Y -43.308,Z -183.185,A -90.000,B 90.000,C 0.000} C_DIS
LIN {X 70.255,Y -43.308,Z -183.682,A -90.000,B 90.000,C 0.000} C_DIS
LIN {X 69.947,Y -43.308,Z -186.265,A -90.000,B 90.000,C 0.000} C_DIS
LIN {X 69.880,Y -43.308,Z -186.766,A -90.000,B 90.000,C 0.000} C_DIS
LIN {X 69.541,Y -43.308,Z -188.961,A -90.000,B 90.000,C 0.000} C_DIS
LIN {X 69.387,Y -43.308,Z -189.779,A -90.000,B 90.000,C 0.000} C_DIS
LIN {X 69.010,Y -43.308,Z -191.510,A -90.000,B 90.000,C 0.000} C_DIS
LIN {X 68.909,Y -43.308,Z -191.888,A -90.000,B 90.000,C 0.000} C_DIS
LIN {X 68.268,Y -43.308,Z -194.347,A -90.000,B 90.000,C 0.000} C_DIS
LIN {X 68.187,Y -43.308,Z -194.653,A -90.000,B 90.000,C 0.000} C_DIS
LIN {X 68.029,Y -43.308,Z -195.156,A -90.000,B 90.000,C 0.000} C_DIS
LIN {X 67.187,Y -43.308,Z -197.917,A -90.000,B 90.000,C 0.000} C_DIS
LIN {X 66.880,Y -43.308,Z -198.797,A -90.000,B 90.000,C 0.000} C_DIS
LIN {X 65.853,Y -43.308,Z -201.780,A -90.000,B 90.000,C 0.000} C_DIS
LIN {X 65.473,Y -43.308,Z -202.794,A -90.000,B 90.000,C 0.000} C_DIS
LIN {X 64.237,Y -43.308,Z -206.123,A -90.000,B 90.000,C 0.000} C_DIS
LIN {X 63.852,Y -43.308,Z -207.097,A -90.000,B 90.000,C 0.000} C_DIS
LIN {X 62.378,Y -43.308,Z -210.855,A -90.000,B 90.000,C 0.000} C_DIS
LIN {X 62.247,Y -43.308,Z -211.182,A -90.000,B 90.000,C 0.000} C_DIS
LIN {X 61.703,Y -43.308,Z -212.501,A -90.000,B 90.000,C 0.000} C_DIS
LIN {X 60.193,Y -43.308,Z -216.188,A -90.000,B 90.000,C 0.000} C_DIS
LIN {X 58.772,Y -43.308,Z -219.535,A -90.000,B 90.000,C 0.000} C_DIS
LIN {X 57.989,Y -43.308,Z -221.360,A -90.000,B 90.000,C 0.000} C_DIS
LIN {X 55.558,Y -43.308,Z -226.621,A -90.000,B 90.000,C 0.000} C_DIS
LIN {X 54.028,Y -43.308,Z -229.559,A -90.000,B 90.000,C 0.000} C_DIS
LIN {X 52.831,Y -43.308,Z -231.898,A -90.000,B 90.000,C 0.000} C_DIS
LIN {X 52.655,Y -43.308,Z -232.202,A -90.000,B 90.000,C 0.000} C_DIS
LIN {X 50.929,Y -43.308,Z -235.057,A -90.000,B 90.000,C 0.000} C_DIS
LIN {X 49.557,Y -43.308,Z -237.417,A -90.000,B 90.000,C 0.000} C_DIS
LIN {X 47.502,Y -43.308,Z -240.262,A -90.000,B 90.000,C 0.000} C_DIS
LIN {X 46.011,Y -43.308,Z -242.469,A -90.000,B 90.000,C 0.000} C_DIS
LIN {X 45.114,Y -43.308,Z -243.561,A -90.000,B 90.000,C 0.000} C_DIS
LIN {X 45.114,Y -60.000,Z -243.561,A -90.000,B 90.000,C 0.000} C_DIS
LIN {X 78.105,Y -60.000,Z -94.806,A -90.000,B 90.000,C 0.000} C_DIS
LIN {X 78.105,Y -43.877,Z -94.806,A -90.000,B 90.000,C 0.000} C_DIS
LIN {X 77.981,Y -43.898,Z -94.435,A -90.000,B 90.000,C 0.000} C_DIS
LIN {X 77.952,Y -43.903,Z -94.305,A -90.000,B 90.000,C 0.000} C_DIS
LIN {X 77.905,Y -43.909,Z -94.087,A -90.000,B 90.000,C 0.000} C_DIS
LIN {X 77.869,Y -43.907,Z -93.914,A -90.000,B 90.000,C 0.000} C_DIS
LIN {X 77.842,Y -43.906,Z -93.765,A -90.000,B 90.000,C 0.000} C_DIS
LIN {X 77.836,Y -43.907,Z -93.523,A -90.000,B 90.000,C 0.000} C_DIS
LIN {X 77.831,Y -43.901,Z -93.298,A -90.000,B 90.000,C 0.000} C_DIS
LIN {X 77.829,Y -43.899,Z -93.229,A -90.000,B 90.000,C 0.000} C_DIS
LIN {X 78.037,Y -43.909,Z -93.090,A -90.000,B 90.000,C 0.000} C_DIS
LIN {X 78.238,Y -43.918,Z -92.948,A -90.000,B 90.000,C 0.000} C_DIS
LIN {X 78.416,Y -43.928,Z -92.858,A -90.000,B 90.000,C 0.000} C_DIS
LIN {X 78.653,Y -43.940,Z -92.735,A -90.000,B 90.000,C 0.000} C_DIS
LIN {X 78.748,Y -43.943,Z -92.678,A -90.000,B 90.000,C 0.000} C_DIS
LIN {X 78.991,Y -43.943,Z -92.524,A -90.000,B 90.000,C 0.000} C_DIS
LIN {X 79.060,Y -43.943,Z -92.475,A -90.000,B 90.000,C 0.000} C_DIS
LIN {X 79.208,Y -43.943,Z -92.363,A -90.000,B 90.000,C 0.000} C_DIS
LIN {X 79.240,Y -43.943,Z -92.341,A -90.000,B 90.000,C 0.000} C_DIS
LIN {X 79.350,Y -43.950,Z -92.265,A -90.000,B 90.000,C 0.000} C_DIS
LIN {X 79.528,Y -43.953,Z -92.144,A -90.000,B 90.000,C 0.000} C_DIS
LIN {X 79.610,Y -43.954,Z -92.085,A -90.000,B 90.000,C 0.000} C_DIS
LIN {X 79.783,Y -43.956,Z -91.948,A -90.000,B 90.000,C 0.000} C_DIS
LIN {X 79.864,Y -43.956,Z -91.879,A -90.000,B 90.000,C 0.000} C_DIS
LIN {X 80.018,Y -43.964,Z -91.734,A -90.000,B 90.000,C 0.000} C_DIS
LIN {X 80.098,Y -43.968,Z -91.653,A -90.000,B 90.000,C 0.000} C_DIS
LIN {X 80.187,Y -43.971,Z -91.558,A -90.000,B 90.000,C 0.000} C_DIS
LIN {X 80.203,Y -43.972,Z -91.545,A -90.000,B 90.000,C 0.000} C_DIS
LIN {X 80.328,Y -43.974,Z -91.447,A -90.000,B 90.000,C 0.000} C_DIS
LIN {X 80.536,Y -43.979,Z -91.266,A -90.000,B 90.000,C 0.000} C_DIS
LIN {X 80.734,Y -43.981,Z -91.069,A -90.000,B 90.000,C 0.000} C_DIS
LIN {X 81.055,Y -43.983,Z -90.707,A -90.000,B 90.000,C 0.000} C_DIS
LIN {X 81.167,Y -43.986,Z -90.612,A -90.000,B 90.000,C 0.000} C_DIS
LIN {X 81.248,Y -43.984,Z -90.544,A -90.000,B 90.000,C 0.000} C_DIS
LIN {X 81.398,Y -43.974,Z -90.419,A -90.000,B 90.000,C 0.000} C_DIS
LIN {X 81.435,Y -43.971,Z -90.393,A -90.000,B 90.000,C 0.000} C_DIS
LIN {X 81.431,Y -43.980,Z -90.558,A -90.000,B 90.000,C 0.000} C_DIS
LIN {X 81.428,Y -43.985,Z -90.720,A -90.000,B 90.000,C 0.000} C_DIS
LIN {X 81.387,Y -43.989,Z -91.486,A -90.000,B 90.000,C 0.000} C_DIS
LIN {X 81.381,Y -43.990,Z -91.587,A -90.000,B 90.000,C 0.000} C_DIS
LIN {X 81.305,Y -43.996,Z -92.150,A -90.000,B 90.000,C 0.000} C_DIS
LIN {X 81.290,Y -43.995,Z -92.262,A -90.000,B 90.000,C 0.000} C_DIS
LIN {X 81.230,Y -43.985,Z -92.697,A -90.000,B 90.000,C 0.000} C_DIS
LIN {X 81.209,Y -43.983,Z -92.814,A -90.000,B 90.000,C 0.000} C_DIS
LIN {X 81.030,Y -43.978,Z -93.433,A -90.000,B 90.000,C 0.000} C_DIS
LIN {X 80.934,Y -43.976,Z -93.588,A -90.000,B 90.000,C 0.000} C_DIS
LIN {X 80.364,Y -43.993,Z -93.859,A -90.000,B 90.000,C 0.000} C_DIS
LIN {X 80.032,Y -44.002,Z -94.005,A -90.000,B 90.000,C 0.000} C_DIS
LIN {X 79.898,Y -43.999,Z -94.069,A -90.000,B 90.000,C 0.000} C_DIS
LIN {X 79.740,Y -43.992,Z -94.146,A -90.000,B 90.000,C 0.000} C_DIS
LIN {X 79.332,Y -43.961,Z -94.350,A -90.000,B 90.000,C 0.000} C_DIS
LIN {X 79.205,Y -43.958,Z -94.414,A -90.000,B 90.000,C 0.000} C_DIS
LIN {X 79.011,Y -43.940,Z -94.516,A -90.000,B 90.000,C 0.000} C_DIS
LIN {X 78.808,Y -43.924,Z -94.571,A -90.000,B 90.000,C 0.000} C_DIS
LIN {X 78.577,Y -43.903,Z -94.644,A -90.000,B 90.000,C 0.000} C_DIS
LIN {X 78.358,Y -43.894,Z -94.716,A -90.000,B 90.000,C 0.000} C_DIS
LIN {X 78.105,Y -43.877,Z -94.806,A -90.000,B 90.000,C 0.000} C_DIS
LIN {X 78.066,Y -43.889,Z -94.694,A -90.000,B 90.000,C 0.000} C_DIS
LIN {X 77.969,Y -43.898,Z -94.446,A -90.000,B 90.000,C 0.000} C_DIS
LIN {X 77.905,Y -43.905,Z -94.250,A -90.000,B 90.000,C 0.000} C_DIS
LIN {X 77.825,Y -43.908,Z -94.028,A -90.000,B 90.000,C 0.000} C_DIS
LIN {X 77.742,Y -43.904,Z -93.809,A -90.000,B 90.000,C 0.000} C_DIS
LIN {X 77.684,Y -43.898,Z -93.588,A -90.000,B 90.000,C 0.000} C_DIS
LIN {X 77.600,Y -43.892,Z -93.302,A -90.000,B 90.000,C 0.000} C_DIS
LIN {X 77.671,Y -43.889,Z -93.215,A -90.000,B 90.000,C 0.000} C_DIS
LIN {X 77.738,Y -43.886,Z -93.116,A -90.000,B 90.000,C 0.000} C_DIS
LIN {X 77.845,Y -43.881,Z -92.926,A -90.000,B 90.000,C 0.000} C_DIS
LIN {X 77.872,Y -43.880,Z -92.862,A -90.000,B 90.000,C 0.000} C_DIS
LIN {X 77.901,Y -43.877,Z -92.778,A -90.000,B 90.000,C 0.000} C_DIS
LIN {X 77.922,Y -43.874,Z -92.686,A -90.000,B 90.000,C 0.000} C_DIS
LIN {X 77.936,Y -43.870,Z -92.557,A -90.000,B 90.000,C 0.000} C_DIS
LIN {X 77.955,Y -43.867,Z -92.446,A -90.000,B 90.000,C 0.000} C_DIS
LIN {X 77.978,Y -43.859,Z -92.190,A -90.000,B 90.000,C 0.000} C_DIS
LIN {X 77.979,Y -43.855,Z -92.062,A -90.000,B 90.000,C 0.000} C_DIS
LIN {X 78.006,Y -43.851,Z -91.944,A -90.000,B 90.000,C 0.000} C_DIS
LIN {X 78.031,Y -43.846,Z -91.779,A -90.000,B 90.000,C 0.000} C_DIS
LIN {X 78.081,Y -43.840,Z -91.600,A -90.000,B 90.000,C 0.000} C_DIS
LIN {X 78.118,Y -43.835,Z -91.447,A -90.000,B 90.000,C 0.000} C_DIS
LIN {X 78.165,Y -43.830,Z -91.300,A -90.000,B 90.000,C 0.000} C_DIS
LIN {X 78.194,Y -43.828,Z -91.233,A -90.000,B 90.000,C 0.000} C_DIS
LIN {X 78.243,Y -43.825,Z -91.139,A -90.000,B 90.000,C 0.000} C_DIS
LIN {X 78.392,Y -43.816,Z -90.885,A -90.000,B 90.000,C 0.000} C_DIS
LIN {X 78.470,Y -43.811,Z -90.741,A -90.000,B 90.000,C 0.000} C_DIS
LIN {X 78.565,Y -43.805,Z -90.608,A -90.000,B 90.000,C 0.000} C_DIS
LIN {X 78.728,Y -43.797,Z -90.403,A -90.000,B 90.000,C 0.000} C_DIS
LIN {X 78.813,Y -43.792,Z -90.270,A -90.000,B 90.000,C 0.000} C_DIS
LIN {X 78.914,Y -43.786,Z -90.091,A -90.000,B 90.000,C 0.000} C_DIS
LIN {X 79.069,Y -43.779,Z -89.945,A -90.000,B 90.000,C 0.000} C_DIS
LIN {X 79.188,Y -43.774,Z -89.823,A -90.000,B 90.000,C 0.000} C_DIS
LIN {X 79.342,Y -43.767,Z -89.645,A -90.000,B 90.000,C 0.000} C_DIS
LIN {X 79.381,Y -43.761,Z -89.600,A -90.000,B 90.000,C 0.000} C_DIS
LIN {X 79.616,Y -43.765,Z -89.333,A -90.000,B 90.000,C 0.000} C_DIS
LIN {X 79.672,Y -43.764,Z -89.273,A -90.000,B 90.000,C 0.000} C_DIS
LIN {X 80.055,Y -43.764,Z -88.950,A -90.000,B 90.000,C 0.000} C_DIS
LIN {X 80.166,Y -43.760,Z -88.857,A -90.000,B 90.000,C 0.000} C_DIS
LIN {X 80.264,Y -43.757,Z -88.784,A -90.000,B 90.000,C 0.000} C_DIS
LIN {X 80.353,Y -43.755,Z -88.725,A -90.000,B 90.000,C 0.000} C_DIS
LIN {X 80.451,Y -43.751,Z -88.652,A -90.000,B 90.000,C 0.000} C_DIS
LIN {X 80.508,Y -43.748,Z -88.605,A -90.000,B 90.000,C 0.000} C_DIS
LIN {X 80.566,Y -43.748,Z -88.580,A -90.000,B 90.000,C 0.000} C_DIS
LIN {X 80.673,Y -43.753,Z -88.531,A -90.000,B 90.000,C 0.000} C_DIS
LIN {X 80.809,Y -43.758,Z -88.465,A -90.000,B 90.000,C 0.000} C_DIS
LIN {X 80.891,Y -43.759,Z -88.419,A -90.000,B 90.000,C 0.000} C_DIS
LIN {X 80.974,Y -43.758,Z -88.367,A -90.000,B 90.000,C 0.000} C_DIS
LIN {X 81.025,Y -43.755,Z -88.334,A -90.000,B 90.000,C 0.000} C_DIS
LIN {X 81.094,Y -43.749,Z -88.285,A -90.000,B 90.000,C 0.000} C_DIS
LIN {X 81.333,Y -43.724,Z -88.095,A -90.000,B 90.000,C 0.000} C_DIS
LIN {X 81.616,Y -43.717,Z -87.885,A -90.000,B 90.000,C 0.000} C_DIS
LIN {X 81.851,Y -43.727,Z -87.815,A -90.000,B 90.000,C 0.000} C_DIS
LIN {X 82.029,Y -43.726,Z -87.764,A -90.000,B 90.000,C 0.000} C_DIS
LIN {X 82.230,Y -43.718,Z -87.708,A -90.000,B 90.000,C 0.000} C_DIS
LIN {X 82.441,Y -43.704,Z -87.650,A -90.000,B 90.000,C 0.000} C_DIS
LIN {X 82.645,Y -43.684,Z -87.596,A -90.000,B 90.000,C 0.000} C_DIS
LIN {X 82.705,Y -43.676,Z -87.580,A -90.000,B 90.000,C 0.000} C_DIS
LIN {X 82.968,Y -43.662,Z -87.672,A -90.000,B 90.000,C 0.000} C_DIS
LIN {X 83.005,Y -43.669,Z -87.790,A -90.000,B 90.000,C 0.000} C_DIS
LIN {X 83.332,Y -43.721,Z -88.784,A -90.000,B 90.000,C 0.000} C_DIS
LIN {X 83.360,Y -43.737,Z -89.016,A -90.000,B 90.000,C 0.000} C_DIS
LIN {X 83.380,Y -43.756,Z -89.296,A -90.000,B 90.000,C 0.000} C_DIS
LIN {X 83.403,Y -43.776,Z -89.643,A -90.000,B 90.000,C 0.000} C_DIS
LIN {X 83.419,Y -43.780,Z -89.916,A -90.000,B 90.000,C 0.000} C_DIS
LIN {X 83.432,Y -43.779,Z -90.153,A -90.000,B 90.000,C 0.000} C_DIS
LIN {X 83.416,Y -43.786,Z -90.795,A -90.000,B 90.000,C 0.000} C_DIS
LIN {X 83.392,Y -43.793,Z -91.286,A -90.000,B 90.000,C 0.000} C_DIS
LIN {X 83.383,Y -43.792,Z -91.452,A -90.000,B 90.000,C 0.000} C_DIS
LIN {X 83.364,Y -43.787,Z -91.759,A -90.000,B 90.000,C 0.000} C_DIS
LIN {X 83.362,Y -43.786,Z -91.789,A -90.000,B 90.000,C 0.000} C_DIS
LIN {X 83.215,Y -43.779,Z -92.865,A -90.000,B 90.000,C 0.000} C_DIS
LIN {X 83.193,Y -43.775,Z -93.015,A -90.000,B 90.000,C 0.000} C_DIS
LIN {X 83.160,Y -43.770,Z -93.204,A -90.000,B 90.000,C 0.000} C_DIS
LIN {X 83.135,Y -43.767,Z -93.313,A -90.000,B 90.000,C 0.000} C_DIS
LIN {X 82.875,Y -43.752,Z -94.208,A -90.000,B 90.000,C 0.000} C_DIS
LIN {X 82.861,Y -43.752,Z -94.248,A -90.000,B 90.000,C 0.000} C_DIS
LIN {X 82.748,Y -43.755,Z -94.434,A -90.000,B 90.000,C 0.000} C_DIS
LIN {X 82.417,Y -43.744,Z -94.965,A -90.000,B 90.000,C 0.000} C_DIS
LIN {X 82.024,Y -43.767,Z -95.270,A -90.000,B 90.000,C 0.000} C_DIS
LIN {X 81.978,Y -43.771,Z -95.293,A -90.000,B 90.000,C 0.000} C_DIS
LIN {X 81.785,Y -43.780,Z -95.387,A -90.000,B 90.000,C 0.000} C_DIS
LIN {X 81.400,Y -43.785,Z -95.570,A -90.000,B 90.000,C 0.000} C_DIS
LIN {X 81.175,Y -43.782,Z -95.675,A -90.000,B 90.000,C 0.000} C_DIS
LIN {X 80.849,Y -43.777,Z -95.817,A -90.000,B 90.000,C 0.000} C_DIS
LIN {X 80.704,Y -43.773,Z -95.886,A -90.000,B 90.000,C 0.000} C_DIS
LIN {X 80.071,Y -43.739,Z -96.204,A -90.000,B 90.000,C 0.000} C_DIS
LIN {X 79.961,Y -43.732,Z -96.264,A -90.000,B 90.000,C 0.000} C_DIS
LIN {X 79.786,Y -43.719,Z -96.371,A -90.000,B 90.000,C 0.000} C_DIS
LIN {X 79.504,Y -43.720,Z -96.441,A -90.000,B 90.000,C 0.000} C_DIS
LIN {X 79.354,Y -43.719,Z -96.485,A -90.000,B 90.000,C 0.000} C_DIS
LIN {X 78.999,Y -43.714,Z -96.602,A -90.000,B 90.000,C 0.000} C_DIS
LIN {X 78.777,Y -43.706,Z -96.681,A -90.000,B 90.000,C 0.000} C_DIS
LIN {X 78.526,Y -43.688,Z -96.772,A -90.000,B 90.000,C 0.000} C_DIS
LIN {X 77.807,Y -43.611,Z -97.019,A -90.000,B 90.000,C 0.000} C_DIS
LIN {X 77.779,Y -43.609,Z -97.026,A -90.000,B 90.000,C 0.000} C_DIS
LIN {X 77.714,Y -43.608,Z -97.004,A -90.000,B 90.000,C 0.000} C_DIS
LIN {X 77.085,Y -43.602,Z -96.813,A -90.000,B 90.000,C 0.000} C_DIS
LIN {X 76.984,Y -43.617,Z -96.676,A -90.000,B 90.000,C 0.000} C_DIS
LIN {X 76.794,Y -43.639,Z -96.418,A -90.000,B 90.000,C 0.000} C_DIS
LIN {X 76.687,Y -43.645,Z -96.270,A -90.000,B 90.000,C 0.000} C_DIS
LIN {X 76.573,Y -43.646,Z -96.112,A -90.000,B 90.000,C 0.000} C_DIS
LIN {X 76.354,Y -43.641,Z -95.806,A -90.000,B 90.000,C 0.000} C_DIS
LIN {X 76.311,Y -43.643,Z -95.698,A -90.000,B 90.000,C 0.000} C_DIS
LIN {X 76.253,Y -43.649,Z -95.535,A -90.000,B 90.000,C 0.000} C_DIS
LIN {X 76.194,Y -43.656,Z -95.358,A -90.000,B 90.000,C 0.000} C_DIS
LIN {X 76.058,Y -43.659,Z -94.941,A -90.000,B 90.000,C 0.000} C_DIS
LIN {X 75.924,Y -43.674,Z -94.317,A -90.000,B 90.000,C 0.000} C_DIS
LIN {X 75.866,Y -43.672,Z -94.002,A -90.000,B 90.000,C 0.000} C_DIS
LIN {X 75.860,Y -43.672,Z -93.953,A -90.000,B 90.000,C 0.000} C_DIS
LIN {X 75.855,Y -43.673,Z -93.764,A -90.000,B 90.000,C 0.000} C_DIS
LIN {X 75.838,Y -43.648,Z -92.989,A -90.000,B 90.000,C 0.000} C_DIS
LIN {X 75.860,Y -43.647,Z -92.831,A -90.000,B 90.000,C 0.000} C_DIS
LIN {X 75.898,Y -43.643,Z -92.557,A -90.000,B 90.000,C 0.000} C_DIS
LIN {X 75.978,Y -43.643,Z -92.405,A -90.000,B 90.000,C 0.000} C_DIS
LIN {X 76.140,Y -43.631,Z -92.102,A -90.000,B 90.000,C 0.000} C_DIS
LIN {X 76.212,Y -43.629,Z -91.949,A -90.000,B 90.000,C 0.000} C_DIS
LIN {X 76.348,Y -43.642,Z -91.847,A -90.000,B 90.000,C 0.000} C_DIS
LIN {X 76.415,Y -43.648,Z -91.790,A -90.000,B 90.000,C 0.000} C_DIS
LIN {X 76.481,Y -43.653,Z -91.729,A -90.000,B 90.000,C 0.000} C_DIS
LIN {X 76.544,Y -43.653,Z -91.667,A -90.000,B 90.000,C 0.000} C_DIS
LIN {X 76.628,Y -43.658,Z -91.627,A -90.000,B 90.000,C 0.000} C_DIS
LIN {X 76.689,Y -43.659,Z -91.595,A -90.000,B 90.000,C 0.000} C_DIS
LIN {X 76.785,Y -43.659,Z -91.540,A -90.000,B 90.000,C 0.000} C_DIS
LIN {X 76.899,Y -43.664,Z -91.463,A -90.000,B 90.000,C 0.000} C_DIS
LIN {X 77.187,Y -43.676,Z -91.260,A -90.000,B 90.000,C 0.000} C_DIS
LIN {X 77.289,Y -43.682,Z -91.202,A -90.000,B 90.000,C 0.000} C_DIS
LIN {X 77.439,Y -43.690,Z -91.126,A -90.000,B 90.000,C 0.000} C_DIS
LIN {X 77.567,Y -43.694,Z -91.063,A -90.000,B 90.000,C 0.000} C_DIS
LIN {X 77.692,Y -43.696,Z -90.998,A -90.000,B 90.000,C 0.000} C_DIS
LIN {X 77.874,Y -43.697,Z -90.883,A -90.000,B 90.000,C 0.000} C_DIS
LIN {X 78.047,Y -43.703,Z -90.751,A -90.000,B 90.000,C 0.000} C_DIS
LIN {X 78.413,Y -43.713,Z -90.501,A -90.000,B 90.000,C 0.000} C_DIS
LIN {X 78.543,Y -43.724,Z -90.396,A -90.000,B 90.000,C 0.000} C_DIS
LIN {X 78.656,Y -43.732,Z -90.288,A -90.000,B 90.000,C 0.000} C_DIS
LIN {X 78.705,Y -43.733,Z -90.236,A -90.000,B 90.000,C 0.000} C_DIS
LIN {X 78.851,Y -43.731,Z -90.066,A -90.000,B 90.000,C 0.000} C_DIS
LIN {X 78.942,Y -43.740,Z -90.004,A -90.000,B 90.000,C 0.000} C_DIS
LIN {X 79.029,Y -43.748,Z -89.941,A -90.000,B 90.000,C 0.000} C_DIS
LIN {X 79.080,Y -43.751,Z -89.900,A -90.000,B 90.000,C 0.000} C_DIS
LIN {X 79.185,Y -43.756,Z -89.809,A -90.000,B 90.000,C 0.000} C_DIS
LIN {X 79.296,Y -43.760,Z -89.697,A -90.000,B 90.000,C 0.000} C_DIS
LIN {X 79.381,Y -43.761,Z -89.600,A -90.000,B 90.000,C 0.000} C_DIS
LIN {X 79.432,Y -43.769,Z -89.540,A -90.000,B 90.000,C 0.000} C_DIS
LIN {X 79.528,Y -43.769,Z -89.414,A -90.000,B 90.000,C 0.000} C_DIS
LIN {X 79.639,Y -43.764,Z -89.249,A -90.000,B 90.000,C 0.000} C_DIS
LIN {X 79.756,Y -43.755,Z -89.092,A -90.000,B 90.000,C 0.000} C_DIS
LIN {X 79.843,Y -43.746,Z -88.961,A -90.000,B 90.000,C 0.000} C_DIS
LIN {X 79.925,Y -43.736,Z -88.824,A -90.000,B 90.000,C 0.000} C_DIS
LIN {X 80.098,Y -43.711,Z -88.513,A -90.000,B 90.000,C 0.000} C_DIS
LIN {X 80.152,Y -43.702,Z -88.405,A -90.000,B 90.000,C 0.000} C_DIS
LIN {X 80.188,Y -43.695,Z -88.321,A -90.000,B 90.000,C 0.000} C_DIS
LIN {X 80.263,Y -43.685,Z -88.204,A -90.000,B 90.000,C 0.000} C_DIS
LIN {X 80.319,Y -43.677,Z -88.105,A -90.000,B 90.000,C 0.000} C_DIS
LIN {X 80.369,Y -43.667,Z -87.998,A -90.000,B 90.000,C 0.000} C_DIS
LIN {X 80.633,Y -43.588,Z -87.385,A -90.000,B 90.000,C 0.000} C_DIS
LIN {X 80.731,Y -43.552,Z -87.097,A -90.000,B 90.000,C 0.000} C_DIS
LIN {X 80.999,Y -43.478,Z -86.535,A -90.000,B 90.000,C 0.000} C_DIS
LIN {X 81.080,Y -43.461,Z -86.410,A -90.000,B 90.000,C 0.000} C_DIS
LIN {X 81.133,Y -43.450,Z -86.335,A -90.000,B 90.000,C 0.000} C_DIS
LIN {X 81.265,Y -43.427,Z -86.200,A -90.000,B 90.000,C 0.000} C_DIS
LIN {X 81.421,Y -43.404,Z -86.074,A -90.000,B 90.000,C 0.000} C_DIS
LIN {X 81.530,Y -43.388,Z -85.997,A -90.000,B 90.000,C 0.000} C_DIS
LIN {X 81.709,Y -43.363,Z -85.884,A -90.000,B 90.000,C 0.000} C_DIS
LIN {X 81.840,Y -43.345,Z -85.814,A -90.000,B 90.000,C 0.000} C_DIS
LIN {X 81.981,Y -43.327,Z -85.751,A -90.000,B 90.000,C 0.000} C_DIS
LIN {X 82.129,Y -43.308,Z -85.700,A -90.000,B 90.000,C 0.000} C_DIS
LIN {X 82.331,Y -43.308,Z -85.642,A -90.000,B 90.000,C 0.000} C_DIS
LIN {X 82.597,Y -43.308,Z -85.582,A -90.000,B 90.000,C 0.000} C_DIS
LIN {X 82.833,Y -43.308,Z -85.579,A -90.000,B 90.000,C 0.000} C_DIS
LIN {X 83.066,Y -43.308,Z -85.626,A -90.000,B 90.000,C 0.000} C_DIS
LIN {X 83.655,Y -43.308,Z -85.826,A -90.000,B 90.000,C 0.000} C_DIS
LIN {X 83.758,Y -43.308,Z -85.812,A -90.000,B 90.000,C 0.000} C_DIS
LIN {X 83.938,Y -43.308,Z -85.820,A -90.000,B 90.000,C 0.000} C_DIS
LIN {X 84.108,Y -43.308,Z -85.876,A -90.000,B 90.000,C 0.000} C_DIS
LIN {X 84.256,Y -43.308,Z -85.977,A -90.000,B 90.000,C 0.000} C_DIS
LIN {X 84.319,Y -43.308,Z -86.052,A -90.000,B 90.000,C 0.000} C_DIS
LIN {X 84.548,Y -43.308,Z -86.331,A -90.000,B 90.000,C 0.000} C_DIS
LIN {X 84.661,Y -43.308,Z -86.525,A -90.000,B 90.000,C 0.000} C_DIS
LIN {X 84.688,Y -43.308,Z -86.584,A -90.000,B 90.000,C 0.000} C_DIS
LIN {X 84.764,Y -43.308,Z -86.810,A -90.000,B 90.000,C 0.000} C_DIS
LIN {X 84.915,Y -43.308,Z -87.308,A -90.000,B 90.000,C 0.000} C_DIS
LIN {X 85.256,Y -43.308,Z -88.376,A -90.000,B 90.000,C 0.000} C_DIS
LIN {X 85.308,Y -43.308,Z -88.857,A -90.000,B 90.000,C 0.000} C_DIS
LIN {X 85.378,Y -43.308,Z -90.140,A -90.000,B 90.000,C 0.000} C_DIS
LIN {X 85.357,Y -43.308,Z -90.874,A -90.000,B 90.000,C 0.000} C_DIS
LIN {X 85.307,Y -43.308,Z -91.825,A -90.000,B 90.000,C 0.000} C_DIS
LIN {X 85.294,Y -43.308,Z -91.995,A -90.000,B 90.000,C 0.000} C_DIS
LIN {X 85.117,Y -43.308,Z -93.300,A -90.000,B 90.000,C 0.000} C_DIS
LIN {X 85.070,Y -43.308,Z -93.577,A -90.000,B 90.000,C 0.000} C_DIS
LIN {X 85.023,Y -43.308,Z -93.791,A -90.000,B 90.000,C 0.000} C_DIS
LIN {X 84.732,Y -43.308,Z -94.808,A -90.000,B 90.000,C 0.000} C_DIS
LIN {X 84.636,Y -43.308,Z -95.073,A -90.000,B 90.000,C 0.000} C_DIS
LIN {X 84.513,Y -43.308,Z -95.287,A -90.000,B 90.000,C 0.000} C_DIS
LIN {X 84.122,Y -43.308,Z -95.923,A -90.000,B 90.000,C 0.000} C_DIS
LIN {X 83.985,Y -43.308,Z -96.138,A -90.000,B 90.000,C 0.000} C_DIS
LIN {X 83.808,Y -43.308,Z -96.348,A -90.000,B 90.000,C 0.000} C_DIS
LIN {X 83.625,Y -43.308,Z -96.499,A -90.000,B 90.000,C 0.000} C_DIS
LIN {X 83.073,Y -43.308,Z -96.917,A -90.000,B 90.000,C 0.000} C_DIS
LIN {X 83.024,Y -43.308,Z -96.947,A -90.000,B 90.000,C 0.000} C_DIS
LIN {X 82.785,Y -43.308,Z -97.065,A -90.000,B 90.000,C 0.000} C_DIS
LIN {X 81.979,Y -43.308,Z -97.445,A -90.000,B 90.000,C 0.000} C_DIS
LIN {X 81.628,Y -43.308,Z -97.598,A -90.000,B 90.000,C 0.000} C_DIS
LIN {X 81.324,Y -43.308,Z -97.755,A -90.000,B 90.000,C 0.000} C_DIS
LIN {X 80.968,Y -43.308,Z -97.939,A -90.000,B 90.000,C 0.000} C_DIS
LIN {X 80.699,Y -43.308,Z -98.111,A -90.000,B 90.000,C 0.000} C_DIS
LIN {X 80.486,Y -43.308,Z -98.215,A -90.000,B 90.000,C 0.000} C_DIS
LIN {X 79.974,Y -43.308,Z -98.341,A -90.000,B 90.000,C 0.000} C_DIS
LIN {X 79.608,Y -43.308,Z -98.463,A -90.000,B 90.000,C 0.000} C_DIS
LIN {X 79.115,Y -43.308,Z -98.648,A -90.000,B 90.000,C 0.000} C_DIS
LIN {X 78.397,Y -43.308,Z -98.908,A -90.000,B 90.000,C 0.000} C_DIS
LIN {X 78.255,Y -43.308,Z -98.945,A -90.000,B 90.000,C 0.000} C_DIS
LIN {X 77.987,Y -43.308,Z -99.054,A -90.000,B 90.000,C 0.000} C_DIS
LIN {X 77.809,Y -43.308,Z -99.083,A -90.000,B 90.000,C 0.000} C_DIS
LIN {X 77.631,Y -43.308,Z -99.061,A -90.000,B 90.000,C 0.000} C_DIS
LIN {X 77.088,Y -43.308,Z -98.880,A -90.000,B 90.000,C 0.000} C_DIS
LIN {X 76.094,Y -43.308,Z -98.581,A -90.000,B 90.000,C 0.000} C_DIS
LIN {X 75.928,Y -43.308,Z -98.511,A -90.000,B 90.000,C 0.000} C_DIS
LIN {X 75.789,Y -43.308,Z -98.399,A -90.000,B 90.000,C 0.000} C_DIS
LIN {X 75.733,Y -43.308,Z -98.322,A -90.000,B 90.000,C 0.000} C_DIS
LIN {X 74.639,Y -43.308,Z -96.798,A -90.000,B 90.000,C 0.000} C_DIS
LIN {X 74.585,Y -43.308,Z -96.693,A -90.000,B 90.000,C 0.000} C_DIS
LIN {X 74.464,Y -43.308,Z -96.390,A -90.000,B 90.000,C 0.000} C_DIS
LIN {X 74.385,Y -43.308,Z -96.166,A -90.000,B 90.000,C 0.000} C_DIS
LIN {X 74.153,Y -43.308,Z -95.450,A -90.000,B 90.000,C 0.000} C_DIS
LIN {X 73.986,Y -43.308,Z -94.657,A -90.000,B 90.000,C 0.000} C_DIS
LIN {X 73.925,Y -43.308,Z -94.320,A -90.000,B 90.000,C 0.000} C_DIS
LIN {X 73.914,Y -43.308,Z -94.246,A -90.000,B 90.000,C 0.000} C_DIS
LIN {X 73.895,Y -43.308,Z -94.085,A -90.000,B 90.000,C 0.000} C_DIS
LIN {X 73.893,Y -43.308,Z -93.954,A -90.000,B 90.000,C 0.000} C_DIS
LIN {X 73.863,Y -43.308,Z -92.882,A -90.000,B 90.000,C 0.000} C_DIS
LIN {X 73.973,Y -43.308,Z -92.082,A -90.000,B 90.000,C 0.000} C_DIS
LIN {X 74.012,Y -43.308,Z -91.907,A -90.000,B 90.000,C 0.000} C_DIS
LIN {X 74.389,Y -43.308,Z -91.191,A -90.000,B 90.000,C 0.000} C_DIS
LIN {X 74.495,Y -43.308,Z -90.881,A -90.000,B 90.000,C 0.000} C_DIS
LIN {X 74.580,Y -43.308,Z -90.723,A -90.000,B 90.000,C 0.000} C_DIS
LIN {X 74.706,Y -43.308,Z -90.595,A -90.000,B 90.000,C 0.000} C_DIS
LIN {X 75.127,Y -43.308,Z -90.298,A -90.000,B 90.000,C 0.000} C_DIS
LIN {X 75.252,Y -43.308,Z -90.148,A -90.000,B 90.000,C 0.000} C_DIS
LIN {X 75.378,Y -43.308,Z -90.020,A -90.000,B 90.000,C 0.000} C_DIS
LIN {X 75.534,Y -43.308,Z -89.932,A -90.000,B 90.000,C 0.000} C_DIS
LIN {X 75.755,Y -43.308,Z -89.862,A -90.000,B 90.000,C 0.000} C_DIS
LIN {X 76.188,Y -43.308,Z -89.560,A -90.000,B 90.000,C 0.000} C_DIS
LIN {X 76.266,Y -43.308,Z -89.524,A -90.000,B 90.000,C 0.000} C_DIS
LIN {X 76.330,Y -43.308,Z -89.483,A -90.000,B 90.000,C 0.000} C_DIS
LIN {X 76.740,Y -43.308,Z -89.282,A -90.000,B 90.000,C 0.000} C_DIS
LIN {X 76.752,Y -43.308,Z -89.271,A -90.000,B 90.000,C 0.000} C_DIS
LIN {X 76.794,Y -43.308,Z -89.240,A -90.000,B 90.000,C 0.000} C_DIS
LIN {X 76.929,Y -43.308,Z -89.138,A -90.000,B 90.000,C 0.000} C_DIS
LIN {X 77.267,Y -43.308,Z -88.913,A -90.000,B 90.000,C 0.000} C_DIS
LIN {X 77.361,Y -43.308,Z -88.800,A -90.000,B 90.000,C 0.000} C_DIS
LIN {X 77.517,Y -43.308,Z -88.621,A -90.000,B 90.000,C 0.000} C_DIS
LIN {X 77.706,Y -43.308,Z -88.479,A -90.000,B 90.000,C 0.000} C_DIS
LIN {X 77.863,Y -43.308,Z -88.376,A -90.000,B 90.000,C 0.000} C_DIS
LIN {X 78.179,Y -43.308,Z -88.019,A -90.000,B 90.000,C 0.000} C_DIS
LIN {X 78.326,Y -43.308,Z -87.861,A -90.000,B 90.000,C 0.000} C_DIS
LIN {X 78.963,Y -43.308,Z -87.323,A -90.000,B 90.000,C 0.000} C_DIS
LIN {X 79.152,Y -43.308,Z -87.181,A -90.000,B 90.000,C 0.000} C_DIS
LIN {X 79.228,Y -43.308,Z -87.132,A -90.000,B 90.000,C 0.000} C_DIS
LIN {X 79.276,Y -43.308,Z -87.079,A -90.000,B 90.000,C 0.000} C_DIS
LIN {X 79.465,Y -43.308,Z -86.937,A -90.000,B 90.000,C 0.000} C_DIS
LIN {X 79.665,Y -43.308,Z -86.845,A -90.000,B 90.000,C 0.000} C_DIS
LIN {X 79.903,Y -43.308,Z -86.739,A -90.000,B 90.000,C 0.000} C_DIS
LIN {X 80.120,Y -43.308,Z -86.559,A -90.000,B 90.000,C 0.000} C_DIS
LIN {X 80.625,Y -43.308,Z -86.182,A -90.000,B 90.000,C 0.000} C_DIS
LIN {X 80.766,Y -43.308,Z -86.111,A -90.000,B 90.000,C 0.000} C_DIS
LIN {X 80.861,Y -43.308,Z -86.067,A -90.000,B 90.000,C 0.000} C_DIS
LIN {X 81.011,Y -43.308,Z -86.022,A -90.000,B 90.000,C 0.000} C_DIS
LIN {X 82.129,Y -43.308,Z -85.700,A -90.000,B 90.000,C 0.000} C_DIS
LIN {X 82.129,Y -60.000,Z -85.700,A -90.000,B 90.000,C 0.000} C_DIS
LIN {X 100.198,Y -60.000,Z -44.162,A -90.000,B 90.000,C 0.000} C_DIS
LIN {X 100.198,Y -41.308,Z -44.162,A -90.000,B 90.000,C 0.000} C_DIS
LIN {X 101.103,Y -41.310,Z -43.143,A -90.000,B 90.000,C 0.000} C_DIS
LIN {X 101.516,Y -41.312,Z -42.682,A -90.000,B 90.000,C 0.000} C_DIS
LIN {X 102.075,Y -41.321,Z -42.070,A -90.000,B 90.000,C 0.000} C_DIS
LIN {X 102.482,Y -41.332,Z -41.624,A -90.000,B 90.000,C 0.000} C_DIS
LIN {X 102.566,Y -41.335,Z -41.538,A -90.000,B 90.000,C 0.000} C_DIS
LIN {X 103.009,Y -41.352,Z -41.087,A -90.000,B 90.000,C 0.000} C_DIS
LIN {X 103.256,Y -41.365,Z -40.837,A -90.000,B 90.000,C 0.000} C_DIS
LIN {X 103.466,Y -41.373,Z -40.647,A -90.000,B 90.000,C 0.000} C_DIS
LIN {X 103.849,Y -41.397,Z -40.305,A -90.000,B 90.000,C 0.000} C_DIS
LIN {X 104.341,Y -41.430,Z -39.877,A -90.000,B 90.000,C 0.000} C_DIS
LIN {X 104.663,Y -41.451,Z -39.633,A -90.000,B 90.000,C 0.000} C_DIS
LIN {X 105.173,Y -41.493,Z -39.252,A -90.000,B 90.000,C 0.000} C_DIS
LIN {X 105.397,Y -41.513,Z -39.092,A -90.000,B 90.000,C 0.000} C_DIS
LIN {X 105.535,Y -41.522,Z -39.002,A -90.000,B 90.000,C 0.000} C_DIS
LIN {X 105.682,Y -41.532,Z -38.910,A -90.000,B 90.000,C 0.000} C_DIS
LIN {X 106.071,Y -41.565,Z -38.670,A -90.000,B 90.000,C 0.000} C_DIS
LIN {X 106.275,Y -41.586,Z -38.546,A -90.000,B 90.000,C 0.000} C_DIS
LIN {X 106.355,Y -41.592,Z -38.502,A -90.000,B 90.000,C 0.000} C_DIS
LIN {X 106.876,Y -41.633,Z -38.224,A -90.000,B 90.000,C 0.000} C_DIS
LIN {X 107.004,Y -41.640,Z -38.164,A -90.000,B 90.000,C 0.000} C_DIS
LIN {X 107.242,Y -41.662,Z -38.055,A -90.000,B 90.000,C 0.000} C_DIS
LIN {X 107.508,Y -41.691,Z -37.940,A -90.000,B 90.000,C 0.000} C_DIS
LIN {X 107.835,Y -41.720,Z -37.813,A -90.000,B 90.000,C 0.000} C_DIS
LIN {X 108.261,Y -41.750,Z -37.675,A -90.000,B 90.000,C 0.000} C_DIS
LIN {X 108.497,Y -41.775,Z -37.605,A -90.000,B 90.000,C 0.000} C_DIS
LIN {X 108.629,Y -41.786,Z -37.572,A -90.000,B 90.000,C 0.000} C_DIS
LIN {X 108.733,Y -41.797,Z -37.547,A -90.000,B 90.000,C 0.000} C_DIS
LIN {X 108.892,Y -41.811,Z -37.514,A -90.000,B 90.000,C 0.000} C_DIS
LIN {X 109.124,Y -41.835,Z -37.469,A -90.000,B 90.000,C 0.000} C_DIS
LIN {X 109.536,Y -41.864,Z -37.412,A -90.000,B 90.000,C 0.000} C_DIS
LIN {X 109.776,Y -41.882,Z -37.384,A -90.000,B 90.000,C 0.000} C_DIS
LIN {X 109.951,Y -41.889,Z -37.377,A -90.000,B 90.000,C 0.000} C_DIS
LIN {X 110.225,Y -41.909,Z -37.372,A -90.000,B 90.000,C 0.000} C_DIS
LIN {X 110.490,Y -41.923,Z -37.375,A -90.000,B 90.000,C 0.000} C_DIS
LIN {X 110.610,Y -41.935,Z -37.381,A -90.000,B 90.000,C 0.000} C_DIS
LIN {X 110.725,Y -41.948,Z -37.390,A -90.000,B 90.000,C 0.000} C_DIS
LIN {X 110.896,Y -41.963,Z -37.408,A -90.000,B 90.000,C 0.000} C_DIS
LIN {X 111.087,Y -41.976,Z -37.436,A -90.000,B 90.000,C 0.000} C_DIS
LIN {X 111.417,Y -42.001,Z -37.494,A -90.000,B 90.000,C 0.000} C_DIS
LIN {X 111.524,Y -42.004,Z -37.519,A -90.000,B 90.000,C 0.000} C_DIS
LIN {X 111.651,Y -42.012,Z -37.553,A -90.000,B 90.000,C 0.000} C_DIS
LIN {X 111.881,Y -42.031,Z -37.622,A -90.000,B 90.000,C 0.000} C_DIS
LIN {X 111.978,Y -42.036,Z -37.654,A -90.000,B 90.000,C 0.000} C_DIS
LIN {X 112.116,Y -42.043,Z -37.707,A -90.000,B 90.000,C 0.000} C_DIS
LIN {X 112.258,Y -42.053,Z -37.765,A -90.000,B 90.000,C 0.000} C_DIS
LIN {X 112.395,Y -42.062,Z -37.832,A -90.000,B 90.000,C 0.000} C_DIS
LIN {X 112.660,Y -42.073,Z -37.971,A -90.000,B 90.000,C 0.000} C_DIS
LIN {X 112.849,Y -42.086,Z -38.083,A -90.000,B 90.000,C 0.000} C_DIS
LIN {X 113.176,Y -42.112,Z -38.301,A -90.000,B 90.000,C 0.000} C_DIS
LIN {X 113.289,Y -42.113,Z -38.385,A -90.000,B 90.000,C 0.000} C_DIS
LIN {X 113.472,Y -42.123,Z -38.535,A -90.000,B 90.000,C 0.000} C_DIS
LIN {X 113.764,Y -42.130,Z -38.822,A -90.000,B 90.000,C 0.000} C_DIS
LIN {X 113.831,Y -42.134,Z -38.896,A -90.000,B 90.000,C 0.000} C_DIS
LIN {X 113.913,Y -42.141,Z -38.994,A -90.000,B 90.000,C 0.000} C_DIS
LIN {X 114.063,Y -42.147,Z -39.189,A -90.000,B 90.000,C 0.000} C_DIS
LIN {X 114.154,Y -42.152,Z -39.310,A -90.000,B 90.000,C 0.000} C_DIS
LIN {X 114.214,Y -42.154,Z -39.408,A -90.000,B 90.000,C 0.000} C_DIS
LIN {X 114.356,Y -42.162,Z -39.653,A -90.000,B 90.000,C 0.000} C_DIS
LIN {X 114.468,Y -42.169,Z -39.867,A -90.000,B 90.000,C 0.000} C_DIS
LIN {X 114.512,Y -42.170,Z -39.956,A -90.000,B 90.000,C 0.000} C_DIS
LIN {X 114.564,Y -42.171,Z -40.071,A -90.000,B 90.000,C 0.000} C_DIS
LIN {X 114.631,Y -42.174,Z -40.227,A -90.000,B 90.000,C 0.000} C_DIS
LIN {X 114.721,Y -42.175,Z -40.465,A -90.000,B 90.000,C 0.000} C_DIS
LIN {X 114.771,Y -42.179,Z -40.626,A -90.000,B 90.000,C 0.000} C_DIS
LIN {X 114.828,Y -42.188,Z -40.840,A -90.000,B 90.000,C 0.000} C_DIS
LIN {X 114.882,Y -42.192,Z -41.080,A -90.000,B 90.000,C 0.000} C_DIS
LIN {X 114.906,Y -42.194,Z -41.215,A -90.000,B 90.000,C 0.000} C_DIS
LIN {X 114.920,Y -42.197,Z -41.303,A -90.000,B 90.000,C 0.000} C_DIS
LIN {X 114.939,Y -42.206,Z -41.461,A -90.000,B 90.000,C 0.000} C_DIS
LIN {X 114.959,Y -42.213,Z -41.685,A -90.000,B 90.000,C 0.000} C_DIS
LIN {X 114.963,Y -42.212,Z -41.743,A -90.000,B 90.000,C 0.000} C_DIS
LIN {X 114.978,Y -42.218,Z -42.066,A -90.000,B 90.000,C 0.000} C_DIS
LIN {X 114.977,Y -42.218,Z -42.145,A -90.000,B 90.000,C 0.000} C_DIS
LIN {X 114.972,Y -42.218,Z -42.278,A -90.000,B 90.000,C 0.000} C_DIS
LIN {X 114.955,Y -42.223,Z -42.495,A -90.000,B 90.000,C 0.000} C_DIS
LIN {X 114.935,Y -42.218,Z -42.667,A -90.000,B 90.000,C 0.000} C_DIS
LIN {X 114.917,Y -42.217,Z -42.793,A -90.000,B 90.000,C 0.000} C_DIS
LIN {X 114.899,Y -42.219,Z -42.892,A -90.000,B 90.000,C 0.000} C_DIS
LIN {X 114.833,Y -42.208,Z -43.173,A -90.000,B 90.000,C 0.000} C_DIS
LIN {X 114.820,Y -42.206,Z -43.224,A -90.000,B 90.000,C 0.000} C_DIS
LIN {X 114.743,Y -42.197,Z -43.513,A -90.000,B 90.000,C 0.000} C_DIS
LIN {X 114.723,Y -42.193,Z -43.576,A -90.000,B 90.000,C 0.000} C_DIS
LIN {X 114.658,Y -42.180,Z -43.763,A -90.000,B 90.000,C 0.000} C_DIS
LIN {X 114.618,Y -42.174,Z -43.871,A -90.000,B 90.000,C 0.000} C_DIS
LIN {X 114.594,Y -42.168,Z -43.930,A -90.000,B 90.000,C 0.000} C_DIS
LIN {X 114.547,Y -42.160,Z -44.037,A -90.000,B 90.000,C 0.000} C_DIS
LIN {X 114.444,Y -42.138,Z -44.276,A -90.000,B 90.000,C 0.000} C_DIS
LIN {X 114.315,Y -42.106,Z -44.569,A -90.000,B 90.000,C 0.000} C_DIS
LIN {X 114.283,Y -42.101,Z -44.644,A -90.000,B 90.000,C 0.000} C_DIS
LIN {X 114.215,Y -42.091,Z -44.808,A -90.000,B 90.000,C 0.000} C_DIS
LIN {X 114.159,Y -42.092,Z -44.968,A -90.000,B 90.000,C 0.000} C_DIS
LIN {X 114.123,Y -42.093,Z -45.079,A -90.000,B 90.000,C 0.000} C_DIS
LIN {X 114.102,Y -42.098,Z -45.158,A -90.000,B 90.000,C 0.000} C_DIS
LIN {X 114.059,Y -42.074,Z -45.576,A -90.000,B 90.000,C 0.000} C_DIS
LIN {X 114.047,Y -42.064,Z -45.704,A -90.000,B 90.000,C 0.000} C_DIS
LIN {X 114.044,Y -42.053,Z -45.856,A -90.000,B 90.000,C 0.000} C_DIS
LIN {X 114.037,Y -42.034,Z -46.048,A -90.000,B 90.000,C 0.000} C_DIS
LIN {X 114.030,Y -42.024,Z -46.169,A -90.000,B 90.000,C 0.000} C_DIS
LIN {X 114.004,Y -42.001,Z -46.479,A -90.000,B 90.000,C 0.000} C_DIS
LIN {X 113.990,Y -41.976,Z -46.704,A -90.000,B 90.000,C 0.000} C_DIS
LIN {X 113.980,Y -41.966,Z -46.811,A -90.000,B 90.000,C 0.000} C_DIS
LIN {X 113.963,Y -41.954,Z -46.958,A -90.000,B 90.000,C 0.000} C_DIS
LIN {X 113.929,Y -41.934,Z -47.252,A -90.000,B 90.000,C 0.000} C_DIS
LIN {X 113.869,Y -41.898,Z -47.706,A -90.000,B 90.000,C 0.000} C_DIS
LIN {X 113.791,Y -41.859,Z -48.118,A -90.000,B 90.000,C 0.000} C_DIS
LIN {X 113.723,Y -41.828,Z -48.468,A -90.000,B 90.000,C 0.000} C_DIS
LIN {X 113.695,Y -41.819,Z -48.595,A -90.000,B 90.000,C 0.000} C_DIS
LIN {X 113.618,Y -41.791,Z -48.904,A -90.000,B 90.000,C 0.000} C_DIS
LIN {X 113.569,Y -41.777,Z -49.093,A -90.000,B 90.000,C 0.000} C_DIS
LIN {X 113.513,Y -41.762,Z -49.292,A -90.000,B 90.000,C 0.000} C_DIS
LIN {X 113.452,Y -41.745,Z -49.505,A -90.000,B 90.000,C 0.000} C_DIS
LIN {X 113.325,Y -41.713,Z -49.923,A -90.000,B 90.000,C 0.000} C_DIS
LIN {X 113.152,Y -41.683,Z -50.457,A -90.000,B 90.000,C 0.000} C_DIS
LIN {X 113.106,Y -41.673,Z -50.580,A -90.000,B 90.000,C 0.000} C_DIS
LIN {X 112.972,Y -41.647,Z -50.928,A -90.000,B 90.000,C 0.000} C_DIS
LIN {X 112.835,Y -41.626,Z -51.277,A -90.000,B 90.000,C 0.000} C_DIS
LIN {X 112.656,Y -41.600,Z -51.727,A -90.000,B 90.000,C 0.000} C_DIS
LIN {X 112.403,Y -41.574,Z -52.335,A -90.000,B 90.000,C 0.000} C_DIS
LIN {X 111.990,Y -41.554,Z -53.316,A -90.000,B 90.000,C 0.000} C_DIS
LIN {X 111.734,Y -41.536,Z -53.898,A -90.000,B 90.000,C 0.000} C_DIS
LIN {X 111.516,Y -41.529,Z -54.423,A -90.000,B 90.000,C 0.000} C_DIS
LIN {X 111.049,Y -41.511,Z -55.530,A -90.000,B 90.000,C 0.000} C_DIS
LIN {X 110.513,Y -41.516,Z -56.889,A -90.000,B 90.000,C 0.000} C_DIS
LIN {X 110.360,Y -41.513,Z -57.270,A -90.000,B 90.000,C 0.000} C_DIS
LIN {X 110.108,Y -41.514,Z -57.957,A -90.000,B 90.000,C 0.000} C_DIS
LIN {X 109.763,Y -41.519,Z -58.891,A -90.000,B 90.000,C 0.000} C_DIS
LIN {X 109.293,Y -41.524,Z -60.256,A -90.000,B 90.000,C 0.000} C_DIS
LIN {X 109.125,Y -41.527,Z -60.736,A -90.000,B 90.000,C 0.000} C_DIS
LIN {X 108.611,Y -41.536,Z -62.232,A -90.000,B 90.000,C 0.000} C_DIS
LIN {X 108.360,Y -41.542,Z -62.958,A -90.000,B 90.000,C 0.000} C_DIS
LIN {X 108.266,Y -41.543,Z -63.222,A -90.000,B 90.000,C 0.000} C_DIS
LIN {X 107.515,Y -41.561,Z -65.313,A -90.000,B 90.000,C 0.000} C_DIS
LIN {X 107.410,Y -41.563,Z -65.589,A -90.000,B 90.000,C 0.000} C_DIS
LIN {X 106.823,Y -41.580,Z -67.085,A -90.000,B 90.000,C 0.000} C_DIS
LIN {X 106.592,Y -41.590,Z -67.655,A -90.000,B 90.000,C 0.000} C_DIS
LIN {X 106.467,Y -41.591,Z -67.946,A -90.000,B 90.000,C 0.000} C_DIS
LIN {X 106.342,Y -41.595,Z -68.229,A -90.000,B 90.000,C 0.000} C_DIS
LIN {X 105.853,Y -41.614,Z -69.338,A -90.000,B 90.000,C 0.000} C_DIS
LIN {X 105.345,Y -41.641,Z -70.447,A -90.000,B 90.000,C 0.000} C_DIS
LIN {X 105.199,Y -41.644,Z -70.750,A -90.000,B 90.000,C 0.000} C_DIS
LIN {X 104.993,Y -41.654,Z -71.170,A -90.000,B 90.000,C 0.000} C_DIS
LIN {X 104.170,Y -41.704,Z -72.784,A -90.000,B 90.000,C 0.000} C_DIS
LIN {X 104.033,Y -41.706,Z -73.034,A -90.000,B 90.000,C 0.000} C_DIS
LIN {X 103.851,Y -41.712,Z -73.356,A -90.000,B 90.000,C 0.000} C_DIS
LIN {X 103.239,Y -41.747,Z -74.421,A -90.000,B 90.000,C 0.000} C_DIS
LIN {X 102.984,Y -41.768,Z -74.857,A -90.000,B 90.000,C 0.000} C_DIS
LIN {X 102.874,Y -41.773,Z -75.036,A -90.000,B 90.000,C 0.000} C_DIS
LIN {X 102.665,Y -41.778,Z -75.364,A -90.000,B 90.000,C 0.000} C_DIS
LIN {X 102.526,Y -41.781,Z -75.577,A -90.000,B 90.000,C 0.000} C_DIS
LIN {X 102.288,Y -41.792,Z -75.929,A -90.000,B 90.000,C 0.000} C_DIS
LIN {X 102.006,Y -41.809,Z -76.342,A -90.000,B 90.000,C 0.000} C_DIS
LIN {X 101.759,Y -41.830,Z -76.692,A -90.000,B 90.000,C 0.000} C_DIS
LIN {X 101.477,Y -41.853,Z -77.087,A -90.000,B 90.000,C 0.000} C_DIS
LIN {X 101.318,Y -41.862,Z -77.302,A -90.000,B 90.000,C 0.000} C_DIS
LIN {X 100.923,Y -41.875,Z -77.813,A -90.000,B 90.000,C 0.000} C_DIS
LIN {X 100.850,Y -41.880,Z -77.904,A -90.000,B 90.000,C 0.000} C_DIS
LIN {X 100.616,Y -41.905,Z -78.182,A -90.000,B 90.000,C 0.000} C_DIS
LIN {X 99.938,Y -41.969,Z -78.975,A -90.000,B 90.000,C 0.000} C_DIS
LIN {X 99.721,Y -41.986,Z -79.223,A -90.000,B 90.000,C 0.000} C_DIS
LIN {X 99.448,Y -42.004,Z -79.528,A -90.000,B 90.000,C 0.000} C_DIS
LIN {X 99.137,Y -42.033,Z -79.860,A -90.000,B 90.000,C 0.000} C_DIS
LIN {X 98.442,Y -42.095,Z -80.559,A -90.000,B 90.000,C 0.000} C_DIS
LIN {X 98.138,Y -42.112,Z -80.852,A -90.000,B 90.000,C 0.000} C_DIS
LIN {X 97.668,Y -42.123,Z -81.265,A -90.000,B 90.000,C 0.000} C_DIS
LIN {X 97.306,Y -42.144,Z -81.561,A -90.000,B 90.000,C 0.000} C_DIS
LIN {X 97.245,Y -42.148,Z -81.610,A -90.000,B 90.000,C 0.000} C_DIS
LIN {X 96.926,Y -42.161,Z -81.847,A -90.000,B 90.000,C 0.000} C_DIS
LIN {X 96.715,Y -42.180,Z -81.988,A -90.000,B 90.000,C 0.000} C_DIS
LIN {X 96.066,Y -42.220,Z -82.398,A -90.000,B 90.000,C 0.000} C_DIS
LIN {X 95.714,Y -42.244,Z -82.615,A -90.000,B 90.000,C 0.000} C_DIS
LIN {X 95.632,Y -42.251,Z -82.664,A -90.000,B 90.000,C 0.000} C_DIS
LIN {X 95.065,Y -42.308,Z -82.982,A -90.000,B 90.000,C 0.000} C_DIS
LIN {X 94.889,Y -42.322,Z -83.077,A -90.000,B 90.000,C 0.000} C_DIS
LIN {X 94.472,Y -42.339,Z -83.294,A -90.000,B 90.000,C 0.000} C_DIS
LIN {X 94.164,Y -42.342,Z -83.448,A -90.000,B 90.000,C 0.000} C_DIS
LIN {X 94.036,Y -42.339,Z -83.510,A -90.000,B 90.000,C 0.000} C_DIS
LIN {X 93.923,Y -42.339,Z -83.560,A -90.000,B 90.000,C 0.000} C_DIS
LIN {X 93.600,Y -42.345,Z -83.690,A -90.000,B 90.000,C 0.000} C_DIS
LIN {X 93.423,Y -42.352,Z -83.753,A -90.000,B 90.000,C 0.000} C_DIS
LIN {X 92.483,Y -42.420,Z -84.031,A -90.000,B 90.000,C 0.000} C_DIS
LIN {X 91.843,Y -42.448,Z -84.209,A -90.000,B 90.000,C 0.000} C_DIS
LIN {X 91.647,Y -42.451,Z -84.258,A -90.000,B 90.000,C 0.000} C_DIS
LIN {X 91.355,Y -42.457,Z -84.325,A -90.000,B 90.000,C 0.000} C_DIS
LIN {X 91.275,Y -42.460,Z -84.342,A -90.000,B 90.000,C 0.000} C_DIS
LIN {X 91.045,Y -42.477,Z -84.381,A -90.000,B 90.000,C 0.000} C_DIS
LIN {X 90.301,Y -42.530,Z -84.517,A -90.000,B 90.000,C 0.000} C_DIS
LIN {X 90.081,Y -42.540,Z -84.554,A -90.000,B 90.000,C 0.000} C_DIS
LIN {X 89.507,Y -42.566,Z -84.647,A -90.000,B 90.000,C 0.000} C_DIS
LIN {X 89.267,Y -42.589,Z -84.688,A -90.000,B 90.000,C 0.000} C_DIS
LIN {X 89.119,Y -42.606,Z -84.704,A -90.000,B 90.000,C 0.000} C_DIS
LIN {X 89.004,Y -42.622,Z -84.710,A -90.000,B 90.000,C 0.000} C_DIS
LIN {X 88.736,Y -42.652,Z -84.743,A -90.000,B 90.000,C 0.000} C_DIS
LIN {X 88.541,Y -42.666,Z -84.767,A -90.000,B 90.000,C 0.000} C_DIS
LIN {X 88.413,Y -42.670,Z -84.794,A -90.000,B 90.000,C 0.000} C_DIS
LIN {X 88.228,Y -42.677,Z -84.827,A -90.000,B 90.000,C 0.000} C_DIS
LIN {X 88.123,Y -42.688,Z -84.848,A -90.000,B 90.000,C 0.000} C_DIS
LIN {X 87.872,Y -42.719,Z -84.881,A -90.000,B 90.000,C 0.000} C_DIS
LIN {X 87.817,Y -42.727,Z -84.884,A -90.000,B 90.000,C 0.000} C_DIS
LIN {X 87.413,Y -42.816,Z -84.906,A -90.000,B 90.000,C 0.000} C_DIS
LIN {X 87.315,Y -42.827,Z -84.905,A -90.000,B 90.000,C 0.000} C_DIS
LIN {X 87.168,Y -42.846,Z -84.896,A -90.000,B 90.000,C 0.000} C_DIS
LIN {X 86.924,Y -42.880,Z -84.865,A -90.000,B 90.000,C 0.000} C_DIS
LIN {X 86.761,Y -42.895,Z -84.864,A -90.000,B 90.000,C 0.000} C_DIS
LIN {X 86.602,Y -42.923,Z -84.865,A -90.000,B 90.000,C 0.000} C_DIS
LIN {X 86.338,Y -42.966,Z -84.866,A -90.000,B 90.000,C 0.000} C_DIS
LIN {X 86.171,Y -42.992,Z -84.858,A -90.000,B 90.000,C 0.000} C_DIS
LIN {X 86.111,Y -43.002,Z -84.852,A -90.000,B 90.000,C 0.000} C_DIS
LIN {X 85.994,Y -43.022,Z -84.835,A -90.000,B 90.000,C 0.000} C_DIS
LIN {X 85.865,Y -43.033,Z -84.813,A -90.000,B 90.000,C 0.000} C_DIS
LIN {X 85.950,Y -43.024,Z -84.919,A -90.000,B 90.000,C 0.000} C_DIS
LIN {X 86.120,Y -42.991,Z -85.137,A -90.000,B 90.000,C 0.000} C_DIS
LIN {X 86.166,Y -42.981,Z -85.202,A -90.000,B 90.000,C 0.000} C_DIS
LIN {X 86.250,Y -42.964,Z -85.339,A -90.000,B 90.000,C 0.000} C_DIS
LIN {X 86.296,Y -42.954,Z -85.423,A -90.000,B 90.000,C 0.000} C_DIS
LIN {X 86.392,Y -42.923,Z -85.600,A -90.000,B 90.000,C 0.000} C_DIS
LIN {X 86.468,Y -42.897,Z -85.769,A -90.000,B 90.000,C 0.000} C_DIS
LIN {X 86.504,Y -42.884,Z -85.860,A -90.000,B 90.000,C 0.000} C_DIS
LIN {X 86.540,Y -42.870,Z -85.967,A -90.000,B 90.000,C 0.000} C_DIS
LIN {X 86.611,Y -42.843,Z -86.202,A -90.000,B 90.000,C 0.000} C_DIS
LIN {X 86.756,Y -42.792,Z -86.720,A -90.000,B 90.000,C 0.000} C_DIS
LIN {X 86.824,Y -42.769,Z -86.954,A -90.000,B 90.000,C 0.000} C_DIS
LIN {X 86.899,Y -42.746,Z -87.213,A -90.000,B 90.000,C 0.000} C_DIS
LIN {X 87.068,Y -42.691,Z -87.798,A -90.000,B 90.000,C 0.000} C_DIS
LIN {X 87.095,Y -42.682,Z -87.901,A -90.000,B 90.000,C 0.000} C_DIS
LIN {X 87.108,Y -42.676,Z -87.964,A -90.000,B 90.000,C 0.000} C_DIS
LIN {X 87.137,Y -42.660,Z -88.171,A -90.000,B 90.000,C 0.000} C_DIS
LIN {X 87.187,Y -42.631,Z -88.754,A -90.000,B 90.000,C 0.000} C_DIS
LIN {X 87.227,Y -42.608,Z -89.642,A -90.000,B 90.000,C 0.000} C_DIS
LIN {X 87.234,Y -42.602,Z -89.810,A -90.000,B 90.000,C 0.000} C_DIS
LIN {X 87.244,Y -42.591,Z -90.194,A -90.000,B 90.000,C 0.000} C_DIS
LIN {X 87.223,Y -42.589,Z -90.927,A -90.000,B 90.000,C 0.000} C_DIS
LIN {X 87.172,Y -42.593,Z -91.924,A -90.000,B 90.000,C 0.000} C_DIS
LIN {X 87.157,Y -42.595,Z -92.139,A -90.000,B 90.000,C 0.000} C_DIS
LIN {X 87.146,Y -42.597,Z -92.245,A -90.000,B 90.000,C 0.000} C_DIS
LIN {X 87.130,Y -42.601,Z -92.373,A -90.000,B 90.000,C 0.000} C_DIS
LIN {X 86.979,Y -42.621,Z -93.551,A -90.000,B 90.000,C 0.000} C_DIS
LIN {X 86.926,Y -42.629,Z -93.882,A -90.000,B 90.000,C 0.000} C_DIS
LIN {X 86.907,Y -42.630,Z -93.983,A -90.000,B 90.000,C 0.000} C_DIS
LIN {X 86.869,Y -42.633,Z -94.160,A -90.000,B 90.000,C 0.000} C_DIS
LIN {X 86.834,Y -42.635,Z -94.309,A -90.000,B 90.000,C 0.000} C_DIS
LIN {X 86.590,Y -42.661,Z -95.192,A -90.000,B 90.000,C 0.000} C_DIS
LIN {X 86.552,Y -42.662,Z -95.328,A -90.000,B 90.000,C 0.000} C_DIS
LIN {X 86.518,Y -42.664,Z -95.436,A -90.000,B 90.000,C 0.000} C_DIS
LIN {X 86.496,Y -42.666,Z -95.498,A -90.000,B 90.000,C 0.000} C_DIS
LIN {X 86.416,Y -42.660,Z -95.716,A -90.000,B 90.000,C 0.000} C_DIS
LIN {X 86.385,Y -42.658,Z -95.794,A -90.000,B 90.000,C 0.000} C_DIS
LIN {X 86.274,Y -42.659,Z -96.019,A -90.000,B 90.000,C 0.000} C_DIS
LIN {X 86.153,Y -42.665,Z -96.234,A -90.000,B 90.000,C 0.000} C_DIS
LIN {X 85.902,Y -42.681,Z -96.653,A -90.000,B 90.000,C 0.000} C_DIS
LIN {X 85.740,Y -42.680,Z -96.916,A -90.000,B 90.000,C 0.000} C_DIS
LIN {X 85.583,Y -42.664,Z -97.153,A -90.000,B 90.000,C 0.000} C_DIS
LIN {X 85.501,Y -42.656,Z -97.268,A -90.000,B 90.000,C 0.000} C_DIS
LIN {X 85.457,Y -42.653,Z -97.322,A -90.000,B 90.000,C 0.000} C_DIS
LIN {X 85.217,Y -42.642,Z -97.601,A -90.000,B 90.000,C 0.000} C_DIS
LIN {X 85.120,Y -42.641,Z -97.702,A -90.000,B 90.000,C 0.000} C_DIS
LIN {X 85.011,Y -42.639,Z -97.798,A -90.000,B 90.000,C 0.000} C_DIS
LIN {X 84.913,Y -42.639,Z -97.880,A -90.000,B 90.000,C 0.000} C_DIS
LIN {X 84.761,Y -42.631,Z -98.000,A -90.000,B 90.000,C 0.000} C_DIS
LIN {X 84.203,Y -42.609,Z -98.411,A -90.000,B 90.000,C 0.000} C_DIS
LIN {X 84.090,Y -42.606,Z -98.490,A -90.000,B 90.000,C 0.000} C_DIS
LIN {X 84.032,Y -42.607,Z -98.526,A -90.000,B 90.000,C 0.000} C_DIS
LIN {X 83.885,Y -42.612,Z -98.613,A -90.000,B 90.000,C 0.000} C_DIS
LIN {X 83.672,Y -42.623,Z -98.722,A -90.000,B 90.000,C 0.000} C_DIS
LIN {X 83.148,Y -42.654,Z -98.983,A -90.000,B 90.000,C 0.000} C_DIS
LIN {X 82.780,Y -42.694,Z -99.171,A -90.000,B 90.000,C 0.000} C_DIS
LIN {X 82.602,Y -42.712,Z -99.256,A -90.000,B 90.000,C 0.000} C_DIS
LIN {X 82.450,Y -42.718,Z -99.324,A -90.000,B 90.000,C 0.000} C_DIS
LIN {X 82.312,Y -42.721,Z -99.397,A -90.000,B 90.000,C 0.000} C_DIS
LIN {X 82.172,Y -42.724,Z -99.470,A -90.000,B 90.000,C 0.000} C_DIS
LIN {X 81.925,Y -42.737,Z -99.602,A -90.000,B 90.000,C 0.000} C_DIS
LIN {X 81.731,Y -42.743,Z -99.728,A -90.000,B 90.000,C 0.000} C_DIS
LIN {X 81.641,Y -42.747,Z -99.783,A -90.000,B 90.000,C 0.000} C_DIS
LIN {X 81.528,Y -42.754,Z -99.844,A -90.000,B 90.000,C 0.000} C_DIS
LIN {X 81.352,Y -42.765,Z -99.934,A -90.000,B 90.000,C 0.000} C_DIS
LIN {X 81.240,Y -42.772,Z -99.988,A -90.000,B 90.000,C 0.000} C_DIS
LIN {X 81.164,Y -42.778,Z -100.020,A -90.000,B 90.000,C 0.000} C_DIS
LIN {X 81.030,Y -42.790,Z -100.068,A -90.000,B 90.000,C 0.000} C_DIS
LIN {X 80.786,Y -42.825,Z -100.139,A -90.000,B 90.000,C 0.000} C_DIS
LIN {X 80.517,Y -42.863,Z -100.215,A -90.000,B 90.000,C 0.000} C_DIS
LIN {X 80.255,Y -42.891,Z -100.309,A -90.000,B 90.000,C 0.000} C_DIS
LIN {X 80.044,Y -42.912,Z -100.393,A -90.000,B 90.000,C 0.000} C_DIS
LIN {X 79.884,Y -42.923,Z -100.456,A -90.000,B 90.000,C 0.000} C_DIS
LIN {X 79.375,Y -42.941,Z -100.645,A -90.000,B 90.000,C 0.000} C_DIS
LIN {X 79.003,Y -42.962,Z -100.782,A -90.000,B 90.000,C 0.000} C_DIS
LIN {X 78.880,Y -42.970,Z -100.819,A -90.000,B 90.000,C 0.000} C_DIS
LIN {X 78.665,Y -42.981,Z -100.907,A -90.000,B 90.000,C 0.000} C_DIS
LIN {X 78.588,Y -42.986,Z -100.934,A -90.000,B 90.000,C 0.000} C_DIS
LIN {X 78.491,Y -42.992,Z -100.964,A -90.000,B 90.000,C 0.000} C_DIS
LIN {X 78.290,Y -42.999,Z -101.007,A -90.000,B 90.000,C 0.000} C_DIS
LIN {X 78.121,Y -43.006,Z -101.035,A -90.000,B 90.000,C 0.000} C_DIS
LIN {X 77.945,Y -43.014,Z -101.056,A -90.000,B 90.000,C 0.000} C_DIS
LIN {X 77.751,Y -43.026,Z -101.062,A -90.000,B 90.000,C 0.000} C_DIS
LIN {X 77.573,Y -43.038,Z -101.050,A -90.000,B 90.000,C 0.000} C_DIS
LIN {X 77.425,Y -43.050,Z -101.034,A -90.000,B 90.000,C 0.000} C_DIS
LIN {X 77.295,Y -43.060,Z -101.017,A -90.000,B 90.000,C 0.000} C_DIS
LIN {X 77.139,Y -43.067,Z -100.984,A -90.000,B 90.000,C 0.000} C_DIS
LIN {X 77.016,Y -43.070,Z -100.949,A -90.000,B 90.000,C 0.000} C_DIS
LIN {X 76.869,Y -43.071,Z -100.900,A -90.000,B 90.000,C 0.000} C_DIS
LIN {X 76.801,Y -43.068,Z -100.877,A -90.000,B 90.000,C 0.000} C_DIS
LIN {X 76.476,Y -43.064,Z -100.768,A -90.000,B 90.000,C 0.000} C_DIS
LIN {X 75.546,Y -43.048,Z -100.487,A -90.000,B 90.000,C 0.000} C_DIS
LIN {X 75.325,Y -43.045,Z -100.408,A -90.000,B 90.000,C 0.000} C_DIS
LIN {X 75.204,Y -43.045,Z -100.357,A -90.000,B 90.000,C 0.000} C_DIS
LIN {X 75.052,Y -43.040,Z -100.289,A -90.000,B 90.000,C 0.000} C_DIS
LIN {X 74.926,Y -43.033,Z -100.220,A -90.000,B 90.000,C 0.000} C_DIS
LIN {X 74.831,Y -43.024,Z -100.159,A -90.000,B 90.000,C 0.000} C_DIS
LIN {X 74.730,Y -43.011,Z -100.084,A -90.000,B 90.000,C 0.000} C_DIS
LIN {X 74.552,Y -42.997,Z -99.939,A -90.000,B 90.000,C 0.000} C_DIS
LIN {X 74.383,Y -42.985,Z -99.785,A -90.000,B 90.000,C 0.000} C_DIS
LIN {X 74.309,Y -42.982,Z -99.704,A -90.000,B 90.000,C 0.000} C_DIS
LIN {X 74.201,Y -42.977,Z -99.569,A -90.000,B 90.000,C 0.000} C_DIS
LIN {X 73.935,Y -42.968,Z -99.197,A -90.000,B 90.000,C 0.000} C_DIS
LIN {X 73.728,Y -42.968,Z -98.909,A -90.000,B 90.000,C 0.000} C_DIS
LIN {X 73.501,Y -42.959,Z -98.590,A -90.000,B 90.000,C 0.000} C_DIS
LIN {X 73.263,Y -42.934,Z -98.250,A -90.000,B 90.000,C 0.000} C_DIS
LIN {X 73.062,Y -42.917,Z -97.965,A -90.000,B 90.000,C 0.000} C_DIS
LIN {X 72.960,Y -42.910,Z -97.810,A -90.000,B 90.000,C 0.000} C_DIS
LIN {X 72.897,Y -42.907,Z -97.695,A -90.000,B 90.000,C 0.000} C_DIS
LIN {X 72.811,Y -42.904,Z -97.523,A -90.000,B 90.000,C 0.000} C_DIS
LIN {X 72.775,Y -42.904,Z -97.442,A -90.000,B 90.000,C 0.000} C_DIS
LIN {X 72.620,Y -42.902,Z -97.050,A -90.000,B 90.000,C 0.000} C_DIS
LIN {X 72.513,Y -42.902,Z -96.740,A -90.000,B 90.000,C 0.000} C_DIS
LIN {X 72.290,Y -42.900,Z -96.054,A -90.000,B 90.000,C 0.000} C_DIS
LIN {X 72.246,Y -42.900,Z -95.896,A -90.000,B 90.000,C 0.000} C_DIS
LIN {X 72.068,Y -42.910,Z -95.061,A -90.000,B 90.000,C 0.000} C_DIS
LIN {X 71.999,Y -42.916,Z -94.691,A -90.000,B 90.000,C 0.000} C_DIS
LIN {X 71.967,Y -42.918,Z -94.480,A -90.000,B 90.000,C 0.000} C_DIS
LIN {X 71.947,Y -42.922,Z -94.317,A -90.000,B 90.000,C 0.000} C_DIS
LIN {X 71.934,Y -42.927,Z -94.185,A -90.000,B 90.000,C 0.000} C_DIS
LIN {X 71.929,Y -42.935,Z -94.038,A -90.000,B 90.000,C 0.000} C_DIS
LIN {X 71.895,Y -42.959,Z -92.937,A -90.000,B 90.000,C 0.000} C_DIS
LIN {X 71.910,Y -42.969,Z -92.615,A -90.000,B 90.000,C 0.000} C_DIS
LIN {X 71.987,Y -43.000,Z -92.019,A -90.000,B 90.000,C 0.000} C_DIS
LIN {X 72.014,Y -43.007,Z -91.814,A -90.000,B 90.000,C 0.000} C_DIS
LIN {X 72.039,Y -43.007,Z -91.670,A -90.000,B 90.000,C 0.000} C_DIS
LIN {X 72.100,Y -43.010,Z -91.400,A -90.000,B 90.000,C 0.000} C_DIS
LIN {X 72.178,Y -43.015,Z -91.163,A -90.000,B 90.000,C 0.000} C_DIS
LIN {X 72.261,Y -43.022,Z -90.984,A -90.000,B 90.000,C 0.000} C_DIS
LIN {X 72.559,Y -43.048,Z -90.410,A -90.000,B 90.000,C 0.000} C_DIS
LIN {X 72.606,Y -43.051,Z -90.275,A -90.000,B 90.000,C 0.000} C_DIS
LIN {X 72.647,Y -43.050,Z -90.160,A -90.000,B 90.000,C 0.000} C_DIS
LIN {X 72.683,Y -43.049,Z -90.073,A -90.000,B 90.000,C 0.000} C_DIS
LIN {X 72.726,Y -43.046,Z -89.984,A -90.000,B 90.000,C 0.000} C_DIS
LIN {X 72.838,Y -43.039,Z -89.778,A -90.000,B 90.000,C 0.000} C_DIS
LIN {X 73.145,Y -43.032,Z -89.358,A -90.000,B 90.000,C 0.000} C_DIS
LIN {X 73.349,Y -43.033,Z -89.152,A -90.000,B 90.000,C 0.000} C_DIS
LIN {X 73.423,Y -43.036,Z -89.085,A -90.000,B 90.000,C 0.000} C_DIS
LIN {X 73.502,Y -43.037,Z -89.021,A -90.000,B 90.000,C 0.000} C_DIS
LIN {X 73.644,Y -43.035,Z -88.919,A -90.000,B 90.000,C 0.000} C_DIS
LIN {X 73.779,Y -43.028,Z -88.826,A -90.000,B 90.000,C 0.000} C_DIS
LIN {X 73.789,Y -43.026,Z -88.814,A -90.000,B 90.000,C 0.000} C_DIS
LIN {X 73.966,Y -43.007,Z -88.636,A -90.000,B 90.000,C 0.000} C_DIS
LIN {X 74.176,Y -42.989,Z -88.454,A -90.000,B 90.000,C 0.000} C_DIS
LIN {X 74.247,Y -42.984,Z -88.403,A -90.000,B 90.000,C 0.000} C_DIS
LIN {X 74.334,Y -42.983,Z -88.346,A -90.000,B 90.000,C 0.000} C_DIS
LIN {X 74.403,Y -42.983,Z -88.305,A -90.000,B 90.000,C 0.000} C_DIS
LIN {X 74.551,Y -42.975,Z -88.222,A -90.000,B 90.000,C 0.000} C_DIS
LIN {X 74.605,Y -42.970,Z -88.193,A -90.000,B 90.000,C 0.000} C_DIS
LIN {X 74.717,Y -42.960,Z -88.140,A -90.000,B 90.000,C 0.000} C_DIS
LIN {X 74.780,Y -42.955,Z -88.113,A -90.000,B 90.000,C 0.000} C_DIS
LIN {X 74.872,Y -42.948,Z -88.079,A -90.000,B 90.000,C 0.000} C_DIS
LIN {X 75.086,Y -42.919,Z -87.937,A -90.000,B 90.000,C 0.000} C_DIS
LIN {X 75.206,Y -42.912,Z -87.863,A -90.000,B 90.000,C 0.000} C_DIS
LIN {X 75.297,Y -42.909,Z -87.814,A -90.000,B 90.000,C 0.000} C_DIS
LIN {X 75.430,Y -42.901,Z -87.744,A -90.000,B 90.000,C 0.000} C_DIS
LIN {X 75.492,Y -42.898,Z -87.714,A -90.000,B 90.000,C 0.000} C_DIS
LIN {X 75.708,Y -42.875,Z -87.613,A -90.000,B 90.000,C 0.000} C_DIS
LIN {X 75.747,Y -42.868,Z -87.587,A -90.000,B 90.000,C 0.000} C_DIS
LIN {X 75.803,Y -42.862,Z -87.547,A -90.000,B 90.000,C 0.000} C_DIS
LIN {X 75.960,Y -42.850,Z -87.445,A -90.000,B 90.000,C 0.000} C_DIS
LIN {X 76.032,Y -42.837,Z -87.366,A -90.000,B 90.000,C 0.000} C_DIS
LIN {X 76.155,Y -42.817,Z -87.241,A -90.000,B 90.000,C 0.000} C_DIS
LIN {X 76.368,Y -42.794,Z -87.067,A -90.000,B 90.000,C 0.000} C_DIS
LIN {X 76.550,Y -42.778,Z -86.936,A -90.000,B 90.000,C 0.000} C_DIS
LIN {X 76.585,Y -42.778,Z -86.910,A -90.000,B 90.000,C 0.000} C_DIS
LIN {X 76.762,Y -42.751,Z -86.721,A -90.000,B 90.000,C 0.000} C_DIS
LIN {X 76.981,Y -42.716,Z -86.505,A -90.000,B 90.000,C 0.000} C_DIS
LIN {X 77.030,Y -42.715,Z -86.458,A -90.000,B 90.000,C 0.000} C_DIS
LIN {X 77.117,Y -42.714,Z -86.382,A -90.000,B 90.000,C 0.000} C_DIS
LIN {X 77.369,Y -42.710,Z -86.171,A -90.000,B 90.000,C 0.000} C_DIS
LIN {X 77.562,Y -42.693,Z -86.016,A -90.000,B 90.000,C 0.000} C_DIS
LIN {X 77.684,Y -42.678,Z -85.919,A -90.000,B 90.000,C 0.000} C_DIS
LIN {X 77.802,Y -42.675,Z -85.822,A -90.000,B 90.000,C 0.000} C_DIS
LIN {X 78.016,Y -42.676,Z -85.661,A -90.000,B 90.000,C 0.000} C_DIS
LIN {X 78.138,Y -42.673,Z -85.562,A -90.000,B 90.000,C 0.000} C_DIS
LIN {X 78.248,Y -42.674,Z -85.479,A -90.000,B 90.000,C 0.000} C_DIS
LIN {X 78.364,Y -42.667,Z -85.396,A -90.000,B 90.000,C 0.000} C_DIS
LIN {X 78.496,Y -42.661,Z -85.312,A -90.000,B 90.000,C 0.000} C_DIS
LIN {X 78.526,Y -42.660,Z -85.295,A -90.000,B 90.000,C 0.000} C_DIS
LIN {X 78.673,Y -42.656,Z -85.220,A -90.000,B 90.000,C 0.000} C_DIS
LIN {X 78.897,Y -42.654,Z -85.118,A -90.000,B 90.000,C 0.000} C_DIS
LIN {X 78.988,Y -42.643,Z -85.050,A -90.000,B 90.000,C 0.000} C_DIS
LIN {X 79.265,Y -42.644,Z -84.843,A -90.000,B 90.000,C 0.000} C_DIS
LIN {X 79.534,Y -42.633,Z -84.648,A -90.000,B 90.000,C 0.000} C_DIS
LIN {X 79.695,Y -42.621,Z -84.551,A -90.000,B 90.000,C 0.000} C_DIS
LIN {X 79.921,Y -42.612,Z -84.437,A -90.000,B 90.000,C 0.000} C_DIS
LIN {X 80.076,Y -42.609,Z -84.365,A -90.000,B 90.000,C 0.000} C_DIS
LIN {X 80.325,Y -42.612,Z -84.270,A -90.000,B 90.000,C 0.000} C_DIS
LIN {X 80.819,Y -42.633,Z -84.119,A -90.000,B 90.000,C 0.000} C_DIS
LIN {X 81.295,Y -42.673,Z -83.967,A -90.000,B 90.000,C 0.000} C_DIS
LIN {X 81.672,Y -42.700,Z -83.849,A -90.000,B 90.000,C 0.000} C_DIS
LIN {X 81.812,Y -42.708,Z -83.806,A -90.000,B 90.000,C 0.000} C_DIS
LIN {X 81.930,Y -42.715,Z -83.775,A -90.000,B 90.000,C 0.000} C_DIS
LIN {X 82.200,Y -42.758,Z -83.700,A -90.000,B 90.000,C 0.000} C_DIS
LIN {X 82.382,Y -42.790,Z -83.662,A -90.000,B 90.000,C 0.000} C_DIS
LIN {X 82.523,Y -42.813,Z -83.646,A -90.000,B 90.000,C 0.000} C_DIS
LIN {X 82.835,Y -42.867,Z -83.629,A -90.000,B 90.000,C 0.000} C_DIS
LIN {X 82.969,Y -42.890,Z -83.628,A -90.000,B 90.000,C 0.000} C_DIS
LIN {X 82.994,Y -42.892,Z -83.630,A -90.000,B 90.000,C 0.000} C_DIS
LIN {X 83.140,Y -42.908,Z -83.644,A -90.000,B 90.000,C 0.000} C_DIS
LIN {X 83.187,Y -42.912,Z -83.651,A -90.000,B 90.000,C 0.000} C_DIS
LIN {X 83.470,Y -42.936,Z -83.703,A -90.000,B 90.000,C 0.000} C_DIS
LIN {X 83.621,Y -42.961,Z -83.737,A -90.000,B 90.000,C 0.000} C_DIS
LIN {X 83.700,Y -42.977,Z -83.759,A -90.000,B 90.000,C 0.000} C_DIS
LIN {X 83.960,Y -43.029,Z -83.839,A -90.000,B 90.000,C 0.000} C_DIS
LIN {X 84.043,Y -43.044,Z -83.840,A -90.000,B 90.000,C 0.000} C_DIS
LIN {X 83.847,Y -42.999,Z -83.693,A -90.000,B 90.000,C 0.000} C_DIS
LIN {X 83.771,Y -42.982,Z -83.633,A -90.000,B 90.000,C 0.000} C_DIS
LIN {X 83.663,Y -42.957,Z -83.535,A -90.000,B 90.000,C 0.000} C_DIS
LIN {X 83.567,Y -42.929,Z -83.434,A -90.000,B 90.000,C 0.000} C_DIS
LIN {X 83.410,Y -42.890,Z -83.256,A -90.000,B 90.000,C 0.000} C_DIS
LIN {X 83.340,Y -42.871,Z -83.172,A -90.000,B 90.000,C 0.000} C_DIS
LIN {X 83.255,Y -42.846,Z -83.056,A -90.000,B 90.000,C 0.000} C_DIS
LIN {X 83.053,Y -42.785,Z -82.750,A -90.000,B 90.000,C 0.000} C_DIS
LIN {X 83.014,Y -42.766,Z -82.686,A -90.000,B 90.000,C 0.000} C_DIS
LIN {X 82.927,Y -42.721,Z -82.524,A -90.000,B 90.000,C 0.000} C_DIS
LIN {X 82.916,Y -42.715,Z -82.500,A -90.000,B 90.000,C 0.000} C_DIS
LIN {X 82.843,Y -42.699,Z -82.354,A -90.000,B 90.000,C 0.000} C_DIS
LIN {X 82.784,Y -42.675,Z -82.228,A -90.000,B 90.000,C 0.000} C_DIS
LIN {X 82.738,Y -42.656,Z -82.122,A -90.000,B 90.000,C 0.000} C_DIS
LIN {X 82.592,Y -42.596,Z -81.734,A -90.000,B 90.000,C 0.000} C_DIS
LIN {X 82.476,Y -42.523,Z -81.397,A -90.000,B 90.000,C 0.000} C_DIS
LIN {X 82.407,Y -42.483,Z -81.240,A -90.000,B 90.000,C 0.000} C_DIS
LIN {X 82.224,Y -42.400,Z -80.840,A -90.000,B 90.000,C 0.000} C_DIS
LIN {X 82.194,Y -42.386,Z -80.769,A -90.000,B 90.000,C 0.000} C_DIS
LIN {X 82.157,Y -42.370,Z -80.675,A -90.000,B 90.000,C 0.000} C_DIS
LIN {X 82.038,Y -42.339,Z -80.332,A -90.000,B 90.000,C 0.000} C_DIS
LIN {X 81.993,Y -42.328,Z -80.195,A -90.000,B 90.000,C 0.000} C_DIS
LIN {X 81.832,Y -42.255,Z -79.524,A -90.000,B 90.000,C 0.000} C_DIS
LIN {X 81.808,Y -42.245,Z -79.410,A -90.000,B 90.000,C 0.000} C_DIS
LIN {X 81.698,Y -42.196,Z -79.016,A -90.000,B 90.000,C 0.000} C_DIS
LIN {X 81.643,Y -42.166,Z -78.869,A -90.000,B 90.000,C 0.000} C_DIS
LIN {X 81.599,Y -42.144,Z -78.739,A -90.000,B 90.000,C 0.000} C_DIS
LIN {X 81.569,Y -42.138,Z -78.650,A -90.000,B 90.000,C 0.000} C_DIS
LIN {X 81.537,Y -42.132,Z -78.547,A -90.000,B 90.000,C 0.000} C_DIS
LIN {X 81.464,Y -42.116,Z -78.308,A -90.000,B 90.000,C 0.000} C_DIS
LIN {X 81.346,Y -42.090,Z -77.867,A -90.000,B 90.000,C 0.000} C_DIS
LIN {X 81.309,Y -42.078,Z -77.719,A -90.000,B 90.000,C 0.000} C_DIS
LIN {X 81.267,Y -42.067,Z -77.519,A -90.000,B 90.000,C 0.000} C_DIS
LIN {X 81.249,Y -42.060,Z -77.422,A -90.000,B 90.000,C 0.000} C_DIS
LIN {X 81.231,Y -42.048,Z -77.351,A -90.000,B 90.000,C 0.000} C_DIS
LIN {X 81.205,Y -42.037,Z -77.259,A -90.000,B 90.000,C 0.000} C_DIS
LIN {X 81.050,Y -41.975,Z -76.720,A -90.000,B 90.000,C 0.000} C_DIS
LIN {X 80.961,Y -41.962,Z -76.447,A -90.000,B 90.000,C 0.000} C_DIS
LIN {X 80.924,Y -41.955,Z -76.314,A -90.000,B 90.000,C 0.000} C_DIS
LIN {X 80.769,Y -41.938,Z -75.693,A -90.000,B 90.000,C 0.000} C_DIS
LIN {X 80.715,Y -41.917,Z -75.414,A -90.000,B 90.000,C 0.000} C_DIS
LIN {X 80.677,Y -41.896,Z -75.262,A -90.000,B 90.000,C 0.000} C_DIS
LIN {X 80.486,Y -41.832,Z -74.591,A -90.000,B 90.000,C 0.000} C_DIS
LIN {X 80.453,Y -41.823,Z -74.464,A -90.000,B 90.000,C 0.000} C_DIS
LIN {X 80.371,Y -41.813,Z -74.121,A -90.000,B 90.000,C 0.000} C_DIS
LIN {X 80.260,Y -41.800,Z -73.635,A -90.000,B 90.000,C 0.000} C_DIS
LIN {X 80.203,Y -41.776,Z -73.293,A -90.000,B 90.000,C 0.000} C_DIS
LIN {X 80.183,Y -41.763,Z -73.199,A -90.000,B 90.000,C 0.000} C_DIS
LIN {X 80.155,Y -41.746,Z -73.053,A -90.000,B 90.000,C 0.000} C_DIS
LIN {X 80.007,Y -41.693,Z -72.364,A -90.000,B 90.000,C 0.000} C_DIS
LIN {X 79.956,Y -41.683,Z -72.078,A -90.000,B 90.000,C 0.000} C_DIS
LIN {X 79.927,Y -41.675,Z -71.906,A -90.000,B 90.000,C 0.000} C_DIS
LIN {X 79.900,Y -41.670,Z -71.730,A -90.000,B 90.000,C 0.000} C_DIS
LIN {X 79.847,Y -41.649,Z -71.309,A -90.000,B 90.000,C 0.000} C_DIS
LIN {X 79.841,Y -41.643,Z -71.234,A -90.000,B 90.000,C 0.000} C_DIS
LIN {X 79.810,Y -41.619,Z -70.805,A -90.000,B 90.000,C 0.000} C_DIS
LIN {X 79.799,Y -41.601,Z -70.558,A -90.000,B 90.000,C 0.000} C_DIS
LIN {X 79.791,Y -41.589,Z -70.410,A -90.000,B 90.000,C 0.000} C_DIS
LIN {X 79.776,Y -41.555,Z -70.010,A -90.000,B 90.000,C 0.000} C_DIS
LIN {X 79.775,Y -41.546,Z -69.896,A -90.000,B 90.000,C 0.000} C_DIS
LIN {X 79.777,Y -41.516,Z -69.230,A -90.000,B 90.000,C 0.000} C_DIS
LIN {X 79.804,Y -41.488,Z -68.807,A -90.000,B 90.000,C 0.000} C_DIS
LIN {X 79.836,Y -41.476,Z -68.415,A -90.000,B 90.000,C 0.000} C_DIS
LIN {X 79.895,Y -41.454,Z -67.973,A -90.000,B 90.000,C 0.000} C_DIS
LIN {X 80.042,Y -41.428,Z -67.193,A -90.000,B 90.000,C 0.000} C_DIS
LIN {X 80.198,Y -41.396,Z -66.595,A -90.000,B 90.000,C 0.000} C_DIS
LIN {X 80.256,Y -41.385,Z -66.405,A -90.000,B 90.000,C 0.000} C_DIS
LIN {X 80.346,Y -41.374,Z -66.127,A -90.000,B 90.000,C 0.000} C_DIS
LIN {X 80.371,Y -41.371,Z -66.058,A -90.000,B 90.000,C 0.000} C_DIS
LIN {X 80.577,Y -41.345,Z -65.593,A -90.000,B 90.000,C 0.000} C_DIS
LIN {X 80.777,Y -41.330,Z -65.151,A -90.000,B 90.000,C 0.000} C_DIS
LIN {X 81.021,Y -41.320,Z -64.615,A -90.000,B 90.000,C 0.000} C_DIS
LIN {X 81.151,Y -41.317,Z -64.361,A -90.000,B 90.000,C 0.000} C_DIS
LIN {X 81.438,Y -41.313,Z -63.804,A -90.000,B 90.000,C 0.000} C_DIS
LIN {X 81.675,Y -41.311,Z -63.397,A -90.000,B 90.000,C 0.000} C_DIS
LIN {X 82.376,Y -41.309,Z -62.271,A -90.000,B 90.000,C 0.000} C_DIS
LIN {X 82.642,Y -41.316,Z -61.843,A -90.000,B 90.000,C 0.000} C_DIS
LIN {X 82.683,Y -41.308,Z -61.777,A -90.000,B 90.000,C 0.000} C_DIS
LIN {X 82.700,Y -41.302,Z -61.748,A -90.000,B 90.000,C 0.000} C_DIS
LIN {X 82.720,Y -41.308,Z -61.722,A -90.000,B 90.000,C 0.000} C_DIS
LIN {X 82.787,Y -41.328,Z -61.629,A -90.000,B 90.000,C 0.000} C_DIS
LIN {X 82.929,Y -41.309,Z -61.435,A -90.000,B 90.000,C 0.000} C_DIS
LIN {X 82.946,Y -41.308,Z -61.410,A -90.000,B 90.000,C 0.000} C_DIS
LIN {X 83.239,Y -41.303,Z -60.998,A -90.000,B 90.000,C 0.000} C_DIS
LIN {X 83.542,Y -41.308,Z -60.592,A -90.000,B 90.000,C 0.000} C_DIS
LIN {X 83.703,Y -41.308,Z -60.371,A -90.000,B 90.000,C 0.000} C_DIS
LIN {X 83.934,Y -41.307,Z -60.043,A -90.000,B 90.000,C 0.000} C_DIS
LIN {X 84.554,Y -41.308,Z -59.189,A -90.000,B 90.000,C 0.000} C_DIS
LIN {X 84.895,Y -41.308,Z -58.707,A -90.000,B 90.000,C 0.000} C_DIS
LIN {X 85.427,Y -41.308,Z -57.937,A -90.000,B 90.000,C 0.000} C_DIS
LIN {X 85.628,Y -41.308,Z -57.639,A -90.000,B 90.000,C 0.000} C_DIS
LIN {X 85.917,Y -41.308,Z -57.194,A -90.000,B 90.000,C 0.000} C_DIS
LIN {X 86.087,Y -41.308,Z -56.916,A -90.000,B 90.000,C 0.000} C_DIS
LIN {X 86.207,Y -41.308,Z -56.707,A -90.000,B 90.000,C 0.000} C_DIS
LIN {X 86.214,Y -41.308,Z -56.705,A -90.000,B 90.000,C 0.000} C_DIS
LIN {X 86.228,Y -41.308,Z -56.712,A -90.000,B 90.000,C 0.000} C_DIS
LIN {X 86.246,Y -41.308,Z -56.716,A -90.000,B 90.000,C 0.000} C_DIS
LIN {X 86.299,Y -41.308,Z -56.709,A -90.000,B 90.000,C 0.000} C_DIS
LIN {X 86.356,Y -41.308,Z -56.689,A -90.000,B 90.000,C 0.000} C_DIS
LIN {X 86.393,Y -41.308,Z -56.672,A -90.000,B 90.000,C 0.000} C_DIS
LIN {X 86.486,Y -41.308,Z -56.622,A -90.000,B 90.000,C 0.000} C_DIS
LIN {X 86.608,Y -41.308,Z -56.547,A -90.000,B 90.000,C 0.000} C_DIS
LIN {X 86.764,Y -41.308,Z -56.441,A -90.000,B 90.000,C 0.000} C_DIS
LIN {X 86.957,Y -41.308,Z -56.300,A -90.000,B 90.000,C 0.000} C_DIS
LIN {X 87.192,Y -41.308,Z -56.119,A -90.000,B 90.000,C 0.000} C_DIS
LIN {X 87.633,Y -41.308,Z -55.763,A -90.000,B 90.000,C 0.000} C_DIS
LIN {X 88.191,Y -41.308,Z -55.289,A -90.000,B 90.000,C 0.000} C_DIS
LIN {X 88.881,Y -41.308,Z -54.682,A -90.000,B 90.000,C 0.000} C_DIS
LIN {X 89.418,Y -41.307,Z -54.191,A -90.000,B 90.000,C 0.000} C_DIS
LIN {X 89.718,Y -41.308,Z -53.925,A -90.000,B 90.000,C 0.000} C_DIS
LIN {X 89.746,Y -41.308,Z -53.899,A -90.000,B 90.000,C 0.000} C_DIS
LIN {X 90.892,Y -41.308,Z -52.852,A -90.000,B 90.000,C 0.000} C_DIS
LIN {X 90.909,Y -41.308,Z -52.838,A -90.000,B 90.000,C 0.000} C_DIS
LIN {X 90.918,Y -41.308,Z -52.839,A -90.000,B 90.000,C 0.000} C_DIS
LIN {X 90.938,Y -41.308,Z -52.829,A -90.000,B 90.000,C 0.000} C_DIS
LIN {X 90.986,Y -41.308,Z -52.795,A -90.000,B 90.000,C 0.000} C_DIS
LIN {X 91.222,Y -41.308,Z -52.606,A -90.000,B 90.000,C 0.000} C_DIS
LIN {X 91.437,Y -41.308,Z -52.426,A -90.000,B 90.000,C 0.000} C_DIS
LIN {X 91.733,Y -41.307,Z -52.170,A -90.000,B 90.000,C 0.000} C_DIS
LIN {X 92.132,Y -41.308,Z -51.835,A -90.000,B 90.000,C 0.000} C_DIS
LIN {X 92.263,Y -41.308,Z -51.722,A -90.000,B 90.000,C 0.000} C_DIS
LIN {X 93.164,Y -41.308,Z -50.956,A -90.000,B 90.000,C 0.000} C_DIS
LIN {X 93.901,Y -41.308,Z -50.338,A -90.000,B 90.000,C 0.000} C_DIS
LIN {X 94.310,Y -46.259,Z -50.001,A -90.000,B 90.000,C 0.000} C_DIS
LIN {X 94.402,Y -46.304,Z -49.925,A -90.000,B 90.000,C 0.000} C_DIS
LIN {X 94.491,Y -46.337,Z -49.852,A -90.000,B 90.000,C 0.000} C_DIS
LIN {X 94.576,Y -46.365,Z -49.783,A -90.000,B 90.000,C 0.000} C_DIS
LIN {X 94.658,Y -46.389,Z -49.717,A -90.000,B 90.000,C 0.000} C_DIS
LIN {X 94.951,Y -46.464,Z -49.484,A -90.000,B 90.000,C 0.000} C_DIS
LIN {X 95.298,Y -46.552,Z -49.216,A -90.000,B 90.000,C 0.000} C_DIS
LIN {X 95.474,Y -46.607,Z -49.086,A -90.000,B 90.000,C 0.000} C_DIS
LIN {X 95.611,Y -46.660,Z -48.989,A -90.000,B 90.000,C 0.000} C_DIS
LIN {X 95.715,Y -46.712,Z -48.921,A -90.000,B 90.000,C 0.000} C_DIS
LIN {X 95.756,Y -46.737,Z -48.896,A -90.000,B 90.000,C 0.000} C_DIS
LIN {X 95.818,Y -46.786,Z -48.861,A -90.000,B 90.000,C 0.000} C_DIS
LIN {X 95.841,Y -46.809,Z -48.850,A -90.000,B 90.000,C 0.000} C_DIS
LIN {X 95.874,Y -46.852,Z -48.839,A -90.000,B 90.000,C 0.000} C_DIS
LIN {X 95.892,Y -46.889,Z -48.837,A -90.000,B 90.000,C 0.000} C_DIS
LIN {X 95.906,Y -46.940,Z -48.845,A -90.000,B 90.000,C 0.000} C_DIS
LIN {X 95.911,Y -46.949,Z -48.844,A -90.000,B 90.000,C 0.000} C_DIS
LIN {X 95.915,Y -46.949,Z -48.840,A -90.000,B 90.000,C 0.000} C_DIS
LIN {X 95.930,Y -46.937,Z -48.824,A -90.000,B 90.000,C 0.000} C_DIS
LIN {X 95.958,Y -46.907,Z -48.792,A -90.000,B 90.000,C 0.000} C_DIS
LIN {X 96.166,Y -46.673,Z -48.552,A -90.000,B 90.000,C 0.000} C_DIS
LIN {X 96.293,Y -46.528,Z -48.409,A -90.000,B 90.000,C 0.000} C_DIS
LIN {X 96.457,Y -46.355,Z -48.226,A -90.000,B 90.000,C 0.000} C_DIS
LIN {X 96.663,Y -46.160,Z -47.999,A -90.000,B 90.000,C 0.000} C_DIS
LIN {X 96.915,Y -45.915,Z -47.722,A -90.000,B 90.000,C 0.000} C_DIS
LIN {X 97.219,Y -45.602,Z -47.393,A -90.000,B 90.000,C 0.000} C_DIS
LIN {X 97.392,Y -45.406,Z -47.206,A -90.000,B 90.000,C 0.000} C_DIS
LIN {X 97.484,Y -45.291,Z -47.107,A -90.000,B 90.000,C 0.000} C_DIS
LIN {X 97.580,Y -45.158,Z -47.004,A -90.000,B 90.000,C 0.000} C_DIS
LIN {X 98.002,Y -44.729,Z -46.553,A -90.000,B 90.000,C 0.000} C_DIS
LIN {X 98.237,Y -44.556,Z -46.303,A -90.000,B 90.000,C 0.000} C_DIS
LIN {X 98.490,Y -44.378,Z -46.034,A -90.000,B 90.000,C 0.000} C_DIS
LIN {X 98.760,Y -44.199,Z -45.748,A -90.000,B 90.000,C 0.000} C_DIS
LIN {X 99.049,Y -41.308,Z -45.443,A -90.000,B 90.000,C 0.000} C_DIS
LIN {X 99.081,Y -41.308,Z -45.409,A -90.000,B 90.000,C 0.000} C_DIS
LIN {X 99.237,Y -44.077,Z -45.244,A -90.000,B 90.000,C 0.000} C_DIS
LIN {X 99.300,Y -44.072,Z -45.178,A -90.000,B 90.000,C 0.000} C_DIS
LIN {X 99.354,Y -44.065,Z -45.121,A -90.000,B 90.000,C 0.000} C_DIS
LIN {X 99.493,Y -44.035,Z -44.973,A -90.000,B 90.000,C 0.000} C_DIS
LIN {X 99.527,Y -44.022,Z -44.937,A -90.000,B 90.000,C 0.000} C_DIS
LIN {X 99.544,Y -44.009,Z -44.918,A -90.000,B 90.000,C 0.000} C_DIS
LIN {X 99.550,Y -43.995,Z -44.910,A -90.000,B 90.000,C 0.000} C_DIS
LIN {X 99.549,Y -43.952,Z -44.906,A -90.000,B 90.000,C 0.000} C_DIS
LIN {X 99.554,Y -43.919,Z -44.897,A -90.000,B 90.000,C 0.000} C_DIS
LIN {X 99.569,Y -43.875,Z -44.877,A -90.000,B 90.000,C 0.000} C_DIS
LIN {X 99.582,Y -43.849,Z -44.860,A -90.000,B 90.000,C 0.000} C_DIS
LIN {X 99.600,Y -43.818,Z -44.839,A -90.000,B 90.000,C 0.000} C_DIS
LIN {X 99.653,Y -43.747,Z -44.776,A -90.000,B 90.000,C 0.000} C_DIS
LIN {X 99.733,Y -43.662,Z -44.685,A -90.000,B 90.000,C 0.000} C_DIS
LIN {X 99.997,Y -41.308,Z -44.389,A -90.000,B 90.000,C 0.000} C_DIS
LIN {X 100.056,Y -41.308,Z -44.323,A -90.000,B 90.000,C 0.000} C_DIS
LIN {X 100.056,Y -60.000,Z -44.323,A -90.000,B 90.000,C 0.000} C_DIS
LIN {X 93.743,Y -60.000,Z -85.432,A -90.000,B 90.000,C 0.000} C_DIS
LIN {X 93.743,Y -41.308,Z -85.432,A -90.000,B 90.000,C 0.000} C_DIS
LIN {X 93.275,Y -41.368,Z -85.586,A -90.000,B 90.000,C 0.000} C_DIS
LIN {X 92.955,Y -41.405,Z -85.689,A -90.000,B 90.000,C 0.000} C_DIS
LIN {X 92.064,Y -41.484,Z -85.958,A -90.000,B 90.000,C 0.000} C_DIS
LIN {X 91.907,Y -41.500,Z -86.002,A -90.000,B 90.000,C 0.000} C_DIS
LIN {X 91.652,Y -41.535,Z -86.075,A -90.000,B 90.000,C 0.000} C_DIS
LIN {X 91.487,Y -41.558,Z -86.114,A -90.000,B 90.000,C 0.000} C_DIS
LIN {X 91.116,Y -41.608,Z -86.191,A -90.000,B 90.000,C 0.000} C_DIS
LIN {X 90.449,Y -41.695,Z -86.332,A -90.000,B 90.000,C 0.000} C_DIS
LIN {X 90.384,Y -41.706,Z -86.347,A -90.000,B 90.000,C 0.000} C_DIS
LIN {X 90.088,Y -41.778,Z -86.421,A -90.000,B 90.000,C 0.000} C_DIS
LIN {X 89.880,Y -41.821,Z -86.468,A -90.000,B 90.000,C 0.000} C_DIS
LIN {X 89.597,Y -41.869,Z -86.527,A -90.000,B 90.000,C 0.000} C_DIS
LIN {X 89.521,Y -41.888,Z -86.544,A -90.000,B 90.000,C 0.000} C_DIS
LIN {X 89.367,Y -41.927,Z -86.573,A -90.000,B 90.000,C 0.000} C_DIS
LIN {X 89.241,Y -41.961,Z -86.593,A -90.000,B 90.000,C 0.000} C_DIS
LIN {X 89.086,Y -42.016,Z -86.616,A -90.000,B 90.000,C 0.000} C_DIS
LIN {X 88.825,Y -42.102,Z -86.667,A -90.000,B 90.000,C 0.000} C_DIS
LIN {X 88.731,Y -42.131,Z -86.694,A -90.000,B 90.000,C 0.000} C_DIS
LIN {X 88.784,Y -42.066,Z -86.930,A -90.000,B 90.000,C 0.000} C_DIS
LIN {X 88.863,Y -41.998,Z -87.254,A -90.000,B 90.000,C 0.000} C_DIS
LIN {X 88.904,Y -41.955,Z -87.455,A -90.000,B 90.000,C 0.000} C_DIS
LIN {X 88.916,Y -41.940,Z -87.529,A -90.000,B 90.000,C 0.000} C_DIS
LIN {X 88.932,Y -41.917,Z -87.654,A -90.000,B 90.000,C 0.000} C_DIS
LIN {X 88.955,Y -41.879,Z -87.885,A -90.000,B 90.000,C 0.000} C_DIS
LIN {X 88.966,Y -41.858,Z -88.046,A -90.000,B 90.000,C 0.000} C_DIS
LIN {X 88.974,Y -41.842,Z -88.182,A -90.000,B 90.000,C 0.000} C_DIS
LIN {X 88.998,Y -41.806,Z -88.556,A -90.000,B 90.000,C 0.000} C_DIS
LIN {X 89.003,Y -41.797,Z -88.655,A -90.000,B 90.000,C 0.000} C_DIS
LIN {X 89.010,Y -41.772,Z -88.996,A -90.000,B 90.000,C 0.000} C_DIS
LIN {X 89.036,Y -41.740,Z -89.706,A -90.000,B 90.000,C 0.000} C_DIS
LIN {X 89.042,Y -41.715,Z -90.178,A -90.000,B 90.000,C 0.000} C_DIS
LIN {X 89.030,Y -41.706,Z -90.500,A -90.000,B 90.000,C 0.000} C_DIS
LIN {X 89.013,Y -41.705,Z -91.030,A -90.000,B 90.000,C 0.000} C_DIS
LIN {X 88.962,Y -41.706,Z -92.018,A -90.000,B 90.000,C 0.000} C_DIS
LIN {X 88.939,Y -41.708,Z -92.333,A -90.000,B 90.000,C 0.000} C_DIS
LIN {X 88.923,Y -41.712,Z -92.491,A -90.000,B 90.000,C 0.000} C_DIS
LIN {X 88.760,Y -41.751,Z -93.817,A -90.000,B 90.000,C 0.000} C_DIS
LIN {X 88.699,Y -41.762,Z -94.207,A -90.000,B 90.000,C 0.000} C_DIS
LIN {X 88.667,Y -41.765,Z -94.375,A -90.000,B 90.000,C 0.000} C_DIS
LIN {X 88.604,Y -41.775,Z -94.669,A -90.000,B 90.000,C 0.000} C_DIS
LIN {X 88.569,Y -41.782,Z -94.819,A -90.000,B 90.000,C 0.000} C_DIS
LIN {X 88.378,Y -41.824,Z -95.549,A -90.000,B 90.000,C 0.000} C_DIS
LIN {X 88.283,Y -41.831,Z -95.888,A -90.000,B 90.000,C 0.000} C_DIS
LIN {X 88.254,Y -41.829,Z -95.975,A -90.000,B 90.000,C 0.000} C_DIS
LIN {X 88.127,Y -41.824,Z -96.328,A -90.000,B 90.000,C 0.000} C_DIS
LIN {X 88.067,Y -41.824,Z -96.483,A -90.000,B 90.000,C 0.000} C_DIS
LIN {X 88.016,Y -41.827,Z -96.598,A -90.000,B 90.000,C 0.000} C_DIS
LIN {X 87.877,Y -41.839,Z -96.890,A -90.000,B 90.000,C 0.000} C_DIS
LIN {X 87.734,Y -41.857,Z -97.153,A -90.000,B 90.000,C 0.000} C_DIS
LIN {X 87.710,Y -41.860,Z -97.196,A -90.000,B 90.000,C 0.000} C_DIS
LIN {X 87.599,Y -41.862,Z -97.377,A -90.000,B 90.000,C 0.000} C_DIS
LIN {X 87.532,Y -41.861,Z -97.485,A -90.000,B 90.000,C 0.000} C_DIS
LIN {X 87.126,Y -41.830,Z -98.115,A -90.000,B 90.000,C 0.000} C_DIS
LIN {X 86.995,Y -41.818,Z -98.300,A -90.000,B 90.000,C 0.000} C_DIS
LIN {X 86.872,Y -41.812,Z -98.459,A -90.000,B 90.000,C 0.000} C_DIS
LIN {X 86.560,Y -41.775,Z -98.803,A -90.000,B 90.000,C 0.000} C_DIS
